KUKA KRL program: EPS_2_251825_SA31_A_20260116064112.src

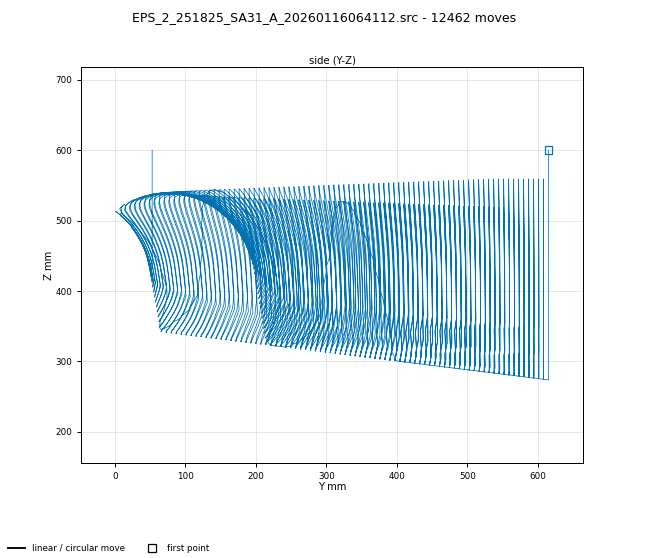
[picture p0: tool path of EPS_2_251825_SA31_A_20260116064112.src, 12462 of 12464 moves have a stored position in this frame; points joined in program order, loops and branches not executed]
&ACCESS RVP
&REL 4
&COMMENT QRS 19112012
&PARAM EDITMASK = *
DEF PART()
EXT BAS (BAS_COMMAND :IN,REAL :IN )
INT I
BAS (#INITMOV,0 )

;KUKA QRS Post kuka4.cps  Date:22-06-2017 !

File_ID=2978

QRS_PRE_INIT()

;Init var - Until changes are made in qrs_pre_init
Outlet_Square_prg=0
Inlet_1_Square_prg=0
Inlet_2_Square_prg=0
Inlet_3_Square_prg=0
Inlet_4_Square_prg=0
Inlet_5_Square_prg=0

Outlet_1={X 0.000, Y 535.490, Z 458.500, B 0.000, E1 0.000 }
Inlet_1={X 0.000, Y 538.340, Z 418.500, B 0.000, E1 227.000 }
Outlet_1_type=201
Inlet_1_type=201
;QRS#1=Sidecore dimensions
;QRS#2=200-8" PVC SDR 35
;QRS#3=200-8" PVC SDR 35
;QRS#4=
;QRS#5=
;QRS#6=
;QRS#7=
;QRS#8=
;QRS#9=12-08 PSX
;QRS#10=12-08 PSX
;QRS#11=
;QRS#12=
;QRS#13=
;QRS#14=
;QRS#15=
;QRS#16=1220x127x838 2,75'
;QRS#17=EPS Height
;QRS#18=559
;QRS#19=*
;QRS#20= UPDATED VERSION 22-06-2017
;QRS#21=*
Outlet_Square=0100
Inlet_1_Square=0100
Inlet_2_Square=0
Inlet_3_Square=0
Inlet_4_Square=0
Inlet_5_Square=0
Mill_Square=1
Outlet_Square_Prg=204
Inlet_1_Square_prg=204

QRS_INIT()

$ADVANCE=5

; T1
PTP {E1 173.626,E2 173.626}
PTP {X 0,Y 615.464,A -85,B 0,C 180,E1 173.626,E2 173.626,E3 0,E4 0,E5 0,E6 0}
QRS_SPEED_INIT()
LIN {X 0,Y 615.464,Z 600,A -85,B 0,C 180,E1 173.626,E2 173.626,E3 0,E4 0,E5 0,E6 0} C_VEL
LIN {X 0,Y 615.464,Z 283.872,A -85,B 0,C 180,E1 173.626,E2 173.626} C_VEL
LIN {X 0,Y 615.464,Z 275.69,A -85,B 0,C 180,E1 173.626,E2 173.626} C_VEL
LIN {X 0,Y 615.457,Z 273.69,A -85,B 0,C 180,E1 173.44,E2 173.44} C_VEL
LIN {X 0,Y 615.487,Z 273.682,A -85,B 0,C 180,E1 170.801,E2 170.801} C_VEL
LIN {X 0,Y 615.492,Z 273.695,A -85,B 0,C 180,E1 168.139,E2 168.139} C_VEL
LIN {X 0,Y 615.46,Z 273.694,A -85,B 0,C 180,E1 165.45,E2 165.45} C_VEL
LIN {X 0,Y 615.46,Z 273.695,A -85,B 0,C 180,E1 163.412,E2 163.412} C_VEL
LIN {X 0,Y 615.46,Z 273.694,A -85,B 0,C 180,E1 161.353,E2 161.353} C_VEL
LIN {X 0,Y 615.458,Z 273.694,A -85,B 0,C 180,E1 159.268,E2 159.268} C_VEL
LIN {X 0,Y 615.455,Z 273.694,A -85,B 0,C 180,E1 157.154,E2 157.154} C_VEL
LIN {X 0,Y 615.451,Z 273.693,A -85,B 0,C 180,E1 155.006,E2 155.006} C_VEL
LIN {X 0,Y 615.448,Z 273.691,A -85,B 0,C 180,E1 152.821,E2 152.821} C_VEL
LIN {X 0,Y 615.475,Z 273.685,A -85,B 0,C 180,E1 150.206,E2 150.206} C_VEL
LIN {X 0,Y 615.493,Z 273.696,A -85,B 0,C 180,E1 147.542,E2 147.542} C_VEL
LIN {X 0,Y 615.481,Z 273.698,A -85,B 0,C 180,E1 145.184,E2 145.184} C_VEL
LIN {X 0,Y 615.45,Z 273.695,A -85,B 0,C 180,E1 142.755,E2 142.755} C_VEL
LIN {X 0,Y 615.446,Z 273.69,A -85,B 0,C 180,E1 140.246,E2 140.246} C_VEL
LIN {X 0,Y 615.491,Z 273.685,A -85,B 0,C 180,E1 137.647,E2 137.647} C_VEL
LIN {X 0,Y 615.483,Z 273.699,A -85,B 0,C 180,E1 134.93,E2 134.93} C_VEL
LIN {X 0,Y 615.442,Z 273.694,A -85,B 0,C 180,E1 132.356,E2 132.356} C_VEL
LIN {X 0,Y 615.438,Z 273.692,A -85,B 0,C 180,E1 130.083,E2 130.083} C_VEL
LIN {X 0,Y 615.437,Z 273.692,A -85,B 0,C 180,E1 128.005,E2 128.005} C_VEL
LIN {X 0,Y 615.449,Z 273.69,A -85,B 0,C 180,E1 125.618,E2 125.618} C_VEL
LIN {X 0,Y 615.474,Z 273.689,A -85,B 0,C 180,E1 123.236,E2 123.236} C_VEL
LIN {X 0,Y 615.491,Z 273.693,A -85,B 0,C 180,E1 120.919,E2 120.919} C_VEL
LIN {X 0,Y 615.435,Z 273.695,A -85,B 0,C 180,E1 117.917,E2 117.917} C_VEL
LIN {X 0,Y 615.433,Z 273.693,A -85,B 0,C 180,E1 115.557,E2 115.557} C_VEL
LIN {X 0,Y 615.484,Z 273.69,A -85,B 0,C 180,E1 112.844,E2 112.844} C_VEL
LIN {X 0,Y 615.454,Z 273.698,A -85,B 0,C 180,E1 110.033,E2 110.033} C_VEL
LIN {X 0,Y 615.452,Z 273.698,A -85,B 0,C 180,E1 107.957,E2 107.957} C_VEL
LIN {X 0,Y 615.451,Z 273.698,A -85,B 0,C 180,E1 105.906,E2 105.906} C_VEL
LIN {X 0,Y 615.454,Z 273.698,A -85,B 0,C 180,E1 103.874,E2 103.874} C_VEL
LIN {X 0,Y 615.458,Z 273.699,A -85,B 0,C 180,E1 101.861,E2 101.861} C_VEL
LIN {X 0,Y 615.423,Z 273.696,A -85,B 0,C 180,E1 99.199,E2 99.199} C_VEL
LIN {X 0,Y 615.421,Z 273.697,A -85,B 0,C 180,E1 97.216,E2 97.216} C_VEL
LIN {X 0,Y 615.423,Z 273.697,A -85,B 0,C 180,E1 95.241,E2 95.241} C_VEL
LIN {X 0,Y 615.426,Z 273.697,A -85,B 0,C 180,E1 93.273,E2 93.273} C_VEL
LIN {X 0,Y 615.431,Z 273.698,A -85,B 0,C 180,E1 91.308,E2 91.308} C_VEL
LIN {X 0,Y 615.433,Z 273.699,A -85,B 0,C 180,E1 89.345,E2 89.345} C_VEL
LIN {X 0,Y 615.446,Z 273.699,A -85,B 0,C 180,E1 87.382,E2 87.382} C_VEL
LIN {X 0,Y 615.415,Z 273.697,A -85,B 0,C 180,E1 84.758,E2 84.758} C_VEL
LIN {X 0,Y 615.414,Z 273.698,A -85,B 0,C 180,E1 82.783,E2 82.783} C_VEL
LIN {X 0,Y 615.415,Z 273.698,A -85,B 0,C 180,E1 80.8,E2 80.8} C_VEL
LIN {X 0,Y 615.416,Z 273.699,A -85,B 0,C 180,E1 78.805,E2 78.805} C_VEL
LIN {X 0,Y 615.418,Z 273.699,A -85,B 0,C 180,E1 76.797,E2 76.797} C_VEL
LIN {X 0,Y 615.419,Z 273.699,A -85,B 0,C 180,E1 74.772,E2 74.772} C_VEL
LIN {X 0,Y 615.419,Z 273.699,A -85,B 0,C 180,E1 72.727,E2 72.727} C_VEL
LIN {X 0,Y 615.418,Z 273.699,A -85,B 0,C 180,E1 70.66,E2 70.66} C_VEL
LIN {X 0,Y 615.414,Z 273.699,A -85,B 0,C 180,E1 68.565,E2 68.565} C_VEL
LIN {X 0,Y 615.408,Z 273.7,A -85,B 0,C 180,E1 66.44,E2 66.44} C_VEL
LIN {X 0,Y 615.405,Z 273.7,A -85,B 0,C 180,E1 64.28,E2 64.28} C_VEL
LIN {X 0,Y 615.402,Z 273.7,A -85,B 0,C 180,E1 62.081,E2 62.081} C_VEL
LIN {X 0,Y 615.423,Z 273.873,A -85,B 0,C 180,E1 61.594,E2 61.594} C_VEL
LIN {X 0,Y 615.459,Z 291.447,A -85,B 0,C 180,E1 58.614,E2 58.614} C_VEL
LIN {X 0,Y 615.456,Z 305.727,A -85,B 0,C 180,E1 56.223,E2 56.223} C_VEL
LIN {X 0,Y 615.472,Z 308.215,A -85,B 0,C 180,E1 55.808,E2 55.808} C_VEL
LIN {X 0,Y 615.477,Z 415.41,A -85,B 0,C 180,E1 54.534,E2 54.534} C_VEL
LIN {X 0,Y 615.47,Z 427.253,A -85,B 0,C 180,E1 54.276,E2 54.276} C_VEL
LIN {X 0,Y 615.484,Z 439.785,A -85,B 0,C 180,E1 53.873,E2 53.873} C_VEL
LIN {X 0,Y 615.479,Z 451.084,A -85,B 0,C 180,E1 53.384,E2 53.384} C_VEL
LIN {X 0,Y 615.493,Z 462.353,A -85,B 0,C 180,E1 52.758,E2 52.758} C_VEL
LIN {X 0,Y 615.495,Z 473.289,A -85,B 0,C 180,E1 51.988,E2 51.988} C_VEL
LIN {X 0,Y 615.496,Z 481.209,A -85,B 0,C 180,E1 51.306,E2 51.306} C_VEL
LIN {X 0,Y 615.499,Z 489.826,A -85,B 0,C 180,E1 50.423,E2 50.423} C_VEL
LIN {X 0,Y 615.49,Z 496.02,A -85,B 0,C 180,E1 49.652,E2 49.652} C_VEL
LIN {X 0,Y 615.495,Z 503.395,A -85,B 0,C 180,E1 48.527,E2 48.527} C_VEL
LIN {X 0,Y 615.495,Z 507.948,A -85,B 0,C 180,E1 47.648,E2 47.648} C_VEL
LIN {X 0,Y 615.498,Z 511.617,A -85,B 0,C 180,E1 46.756,E2 46.756} C_VEL
LIN {X 0,Y 615.498,Z 514.488,A -85,B 0,C 180,E1 45.851,E2 45.851} C_VEL
LIN {X 0,Y 615.496,Z 516.585,A -85,B 0,C 180,E1 44.932,E2 44.932} C_VEL
LIN {X 0,Y 615.495,Z 517.891,A -85,B 0,C 180,E1 43.998,E2 43.998} C_VEL
LIN {X 0,Y 615.496,Z 518.372,A -85,B 0,C 180,E1 43.048,E2 43.048} C_VEL
LIN {X 0,Y 615.498,Z 518.018,A -85,B 0,C 180,E1 42.081,E2 42.081} C_VEL
LIN {X 0,Y 615.495,Z 516.78,A -85,B 0,C 180,E1 41.095,E2 41.095} C_VEL
LIN {X 0,Y 615.493,Z 513.618,A -85,B 0,C 180,E1 39.75,E2 39.75} C_VEL
LIN {X 0,Y 615.493,Z 508.935,A -85,B 0,C 180,E1 38.485,E2 38.485} C_VEL
LIN {X 0,Y 615.497,Z 503.671,A -85,B 0,C 180,E1 37.434,E2 37.434} C_VEL
LIN {X 0,Y 615.493,Z 497.261,A -85,B 0,C 180,E1 36.425,E2 36.425} C_VEL
LIN {X 0,Y 615.493,Z 489.182,A -85,B 0,C 180,E1 35.415,E2 35.415} C_VEL
LIN {X 0,Y 615.494,Z 478.595,A -85,B 0,C 180,E1 34.362,E2 34.362} C_VEL
LIN {X 0,Y 615.497,Z 468.094,A -85,B 0,C 180,E1 33.535,E2 33.535} C_VEL
LIN {X 0,Y 615.46,Z 457.245,A -85,B 0,C 180,E1 32.848,E2 32.848} C_VEL
LIN {X 0,Y 615.493,Z 445.048,A -85,B 0,C 180,E1 32.25,E2 32.25} C_VEL
LIN {X 0,Y 615.466,Z 433.199,A -85,B 0,C 180,E1 31.808,E2 31.808} C_VEL
LIN {X 0,Y 615.439,Z 419.96,A -85,B 0,C 180,E1 31.459,E2 31.459} C_VEL
LIN {X 0,Y 615.434,Z 406.25,A -85,B 0,C 180,E1 31.249,E2 31.249} C_VEL
LIN {X 0,Y 615.497,Z 308.14,A -85,B 0,C 180,E1 30.091,E2 30.091} C_VEL
LIN {X 0,Y 615.466,Z 291.844,A -85,B 0,C 180,E1 27.363,E2 27.363} C_VEL
LIN {X 0,Y 615.481,Z 275.707,A -85,B 0,C 180,E1 24.632,E2 24.632} C_VEL
LIN {X 0,Y 615.473,Z 273.688,A -85,B 0,C 180,E1 24.273,E2 24.273} C_VEL
LIN {X 0,Y 615.474,Z 273.686,A -85,B 0,C 180,E1 22.137,E2 22.137} C_VEL
LIN {X 0,Y 615.48,Z 273.685,A -85,B 0,C 180,E1 19.338,E2 19.338} C_VEL
LIN {X 0,Y 615.482,Z 273.697,A -85,B 0,C 180,E1 16.429,E2 16.429} C_VEL
LIN {X 0,Y 615.474,Z 273.686,A -85,B 0,C 180,E1 13.875,E2 13.875} C_VEL
LIN {X 0,Y 615.486,Z 273.682,A -85,B 0,C 180,E1 11.193,E2 11.193} C_VEL
LIN {X 0,Y 615.483,Z 273.696,A -85,B 0,C 180,E1 8.537,E2 8.537} C_VEL
LIN {X 0,Y 615.475,Z 273.693,A -85,B 0,C 180,E1 5.899,E2 5.899} C_VEL
LIN {X 0,Y 615.485,Z 273.681,A -85,B 0,C 180,E1 3.273,E2 3.273} C_VEL
LIN {X 0,Y 615.477,Z 273.687,A -85,B 0,C 180,E1 0.654,E2 0.654} C_VEL
LIN {X 0,Y 615.497,Z 273.7,A -85,B 0,C 180,E1 -1.963,E2 -1.963} C_VEL
LIN {X 0,Y 615.472,Z 273.69,A -85,B 0,C 180,E1 -4.585,E2 -4.585} C_VEL
LIN {X 0,Y 615.486,Z 273.681,A -85,B 0,C 180,E1 -7.216,E2 -7.216} C_VEL
LIN {X 0,Y 615.479,Z 273.691,A -85,B 0,C 180,E1 -9.862,E2 -9.862} C_VEL
LIN {X 0,Y 615.479,Z 273.697,A -85,B 0,C 180,E1 -12.53,E2 -12.53} C_VEL
LIN {X 0,Y 615.478,Z 273.683,A -85,B 0,C 180,E1 -15.226,E2 -15.226} C_VEL
LIN {X 0,Y 615.478,Z 273.687,A -85,B 0,C 180,E1 -17.957,E2 -17.957} C_VEL
LIN {X 0,Y 615.483,Z 273.699,A -85,B 0,C 180,E1 -20.731,E2 -20.731} C_VEL
LIN {X 0,Y 615.48,Z 273.682,A -85,B 0,C 180,E1 -23.557,E2 -23.557} C_VEL
LIN {X 0,Y 615.481,Z 273.692,A -85,B 0,C 180,E1 -26.444,E2 -26.444} C_VEL
LIN {X 0,Y 615.486,Z 273.695,A -85,B 0,C 180,E1 -28.658,E2 -28.658} C_VEL
LIN {X 0,Y 615.481,Z 273.698,A -85,B 0,C 180,E1 -31.085,E2 -31.085} C_VEL
LIN {X 0,Y 615.489,Z 273.68,A -85,B 0,C 180,E1 -34.022,E2 -34.022} C_VEL
LIN {X 0,Y 615.483,Z 273.696,A -85,B 0,C 180,E1 -36.936,E2 -36.936} C_VEL
LIN {X 0,Y 615.47,Z 273.689,A -85,B 0,C 180,E1 -39.752,E2 -39.752} C_VEL
LIN {X 0,Y 615.493,Z 273.679,A -85,B 0,C 180,E1 -42.353,E2 -42.353} C_VEL
LIN {X 0,Y 615.482,Z 273.692,A -85,B 0,C 180,E1 -45.069,E2 -45.069} C_VEL
LIN {X 0,Y 615.47,Z 273.691,A -85,B 0,C 180,E1 -47.922,E2 -47.922} C_VEL
LIN {X 0,Y 615.471,Z 273.686,A -85,B 0,C 180,E1 -50.248,E2 -50.248} C_VEL
LIN {X 0,Y 615.482,Z 273.686,A -85,B 0,C 180,E1 -53.064,E2 -53.064} C_VEL
LIN {X 0,Y 615.479,Z 273.695,A -85,B 0,C 180,E1 -55.977,E2 -55.977} C_VEL
LIN {X 0,Y 615.469,Z 273.69,A -85,B 0,C 180,E1 -58.313,E2 -58.313} C_VEL
LIN {X 0,Y 615.469,Z 273.687,A -85,B 0,C 180,E1 -60.593,E2 -60.593} C_VEL
LIN {X 0,Y 615.486,Z 273.681,A -85,B 0,C 180,E1 -62.956,E2 -62.956} C_VEL
LIN {X 0,Y 615.481,Z 273.692,A -85,B 0,C 180,E1 -65.727,E2 -65.727} C_VEL
LIN {X 0,Y 615.487,Z 273.753,A -85,B 0,C 180,E1 -67.437,E2 -67.437} C_VEL
LIN {X 0,Y 615.455,Z 293.69,A -85,B 0,C 180,E1 -70.14,E2 -70.14} C_VEL
LIN {X 0,Y 615.472,Z 313.075,A -85,B 0,C 180,E1 -72.729,E2 -72.729} C_VEL
LIN {X 0,Y 615.493,Z 334.915,A -85,B 0,C 180,E1 -75.606,E2 -75.606} C_VEL
LIN {X 0,Y 615.471,Z 346.466,A -85,B 0,C 180,E1 -77.113,E2 -77.113} C_VEL
LIN {X 0,Y 615.457,Z 454.82,A -85,B 0,C 180,E1 -78.41,E2 -78.41} C_VEL
LIN {X 0,Y 615.456,Z 467.338,A -85,B 0,C 180,E1 -78.681,E2 -78.681} C_VEL
LIN {X 0,Y 615.483,Z 480.687,A -85,B 0,C 180,E1 -79.115,E2 -79.115} C_VEL
LIN {X 0,Y 615.492,Z 492.47,A -85,B 0,C 180,E1 -79.639,E2 -79.639} C_VEL
LIN {X 0,Y 615.483,Z 503.991,A -85,B 0,C 180,E1 -80.303,E2 -80.303} C_VEL
LIN {X 0,Y 615.499,Z 514.337,A -85,B 0,C 180,E1 -81.05,E2 -81.05} C_VEL
LIN {X 0,Y 615.497,Z 522.688,A -85,B 0,C 180,E1 -81.794,E2 -81.794} C_VEL
LIN {X 0,Y 615.498,Z 530.603,A -85,B 0,C 180,E1 -82.619,E2 -82.619} C_VEL
LIN {X 0,Y 615.491,Z 538.202,A -85,B 0,C 180,E1 -83.608,E2 -83.608} C_VEL
LIN {X 0,Y 615.498,Z 545.203,A -85,B 0,C 180,E1 -84.759,E2 -84.759} C_VEL
LIN {X 0,Y 615.493,Z 549.85,A -85,B 0,C 180,E1 -85.743,E2 -85.743} C_VEL
LIN {X 0,Y 615.494,Z 553.398,A -85,B 0,C 180,E1 -86.727,E2 -86.727} C_VEL
LIN {X 0,Y 615.497,Z 555.232,A -85,B 0,C 180,E1 -87.382,E2 -87.382} C_VEL
LIN {X 0,Y 615.497,Z 556.607,A -85,B 0,C 180,E1 -88.037,E2 -88.037} C_VEL
LIN {X 0,Y 615.496,Z 558.173,A -85,B 0,C 180,E1 -89.345,E2 -89.345} C_VEL
LIN {X 0,Y 615.494,Z 558.389,A -85,B 0,C 180,E1 -90,E2 -90} C_VEL
LIN {X 0,Y 615.495,Z 557.58,A -85,B 0,C 180,E1 -91.308,E2 -91.308} C_VEL
LIN {X 0,Y 615.497,Z 556.609,A -85,B 0,C 180,E1 -91.963,E2 -91.963} C_VEL
LIN {X 0,Y 615.497,Z 555.234,A -85,B 0,C 180,E1 -92.617,E2 -92.617} C_VEL
LIN {X 0,Y 615.496,Z 552.351,A -85,B 0,C 180,E1 -93.6,E2 -93.6} C_VEL
LIN {X 0,Y 615.498,Z 548.443,A -85,B 0,C 180,E1 -94.584,E2 -94.584} C_VEL
LIN {X 0,Y 615.499,Z 543.407,A -85,B 0,C 180,E1 -95.569,E2 -95.569} C_VEL
LIN {X 0,Y 615.49,Z 536.913,A -85,B 0,C 180,E1 -96.578,E2 -96.578} C_VEL
LIN {X 0,Y 615.497,Z 529.137,A -85,B 0,C 180,E1 -97.545,E2 -97.545} C_VEL
LIN {X 0,Y 615.498,Z 519.262,A -85,B 0,C 180,E1 -98.536,E2 -98.536} C_VEL
LIN {X 0,Y 615.495,Z 508.872,A -85,B 0,C 180,E1 -99.364,E2 -99.364} C_VEL
LIN {X 0,Y 615.482,Z 498.584,A -85,B 0,C 180,E1 -100.028,E2 -100.028} C_VEL
LIN {X 0,Y 615.495,Z 487.144,A -85,B 0,C 180,E1 -100.616,E2 -100.616} C_VEL
LIN {X 0,Y 615.467,Z 475.366,A -85,B 0,C 180,E1 -101.077,E2 -101.077} C_VEL
LIN {X 0,Y 615.455,Z 462.267,A -85,B 0,C 180,E1 -101.443,E2 -101.443} C_VEL
LIN {X 0,Y 615.461,Z 448.986,A -85,B 0,C 180,E1 -101.673,E2 -101.673} C_VEL
LIN {X 0,Y 615.471,Z 346.472,A -85,B 0,C 180,E1 -102.886,E2 -102.886} C_VEL
LIN {X 0,Y 615.455,Z 325.994,A -85,B 0,C 180,E1 -105.566,E2 -105.566} C_VEL
LIN {X 0,Y 615.481,Z 305.476,A -85,B 0,C 180,E1 -108.281,E2 -108.281} C_VEL
LIN {X 0,Y 615.468,Z 283.348,A -85,B 0,C 180,E1 -111.256,E2 -111.256} C_VEL
LIN {X 0,Y 615.489,Z 273.682,A -85,B 0,C 180,E1 -112.594,E2 -112.594} C_VEL
LIN {X 0,Y 615.485,Z 273.681,A -85,B 0,C 180,E1 -114.991,E2 -114.991} C_VEL
LIN {X 0,Y 615.482,Z 273.699,A -85,B 0,C 180,E1 -117.915,E2 -117.915} C_VEL
LIN {X 0,Y 615.485,Z 273.682,A -85,B 0,C 180,E1 -120.919,E2 -120.919} C_VEL
LIN {X 0,Y 615.473,Z 273.686,A -85,B 0,C 180,E1 -123.532,E2 -123.532} C_VEL
LIN {X 0,Y 615.487,Z 273.696,A -85,B 0,C 180,E1 -126.424,E2 -126.424} C_VEL
LIN {X 0,Y 615.48,Z 273.684,A -85,B 0,C 180,E1 -129.061,E2 -129.061} C_VEL
LIN {X 0,Y 615.492,Z 273.68,A -85,B 0,C 180,E1 -131.473,E2 -131.473} C_VEL
LIN {X 0,Y 615.477,Z 273.693,A -85,B 0,C 180,E1 -134.15,E2 -134.15} C_VEL
LIN {X 0,Y 615.476,Z 273.691,A -85,B 0,C 180,E1 -136.953,E2 -136.953} C_VEL
LIN {X 0,Y 615.481,Z 273.683,A -85,B 0,C 180,E1 -139.393,E2 -139.393} C_VEL
LIN {X 0,Y 615.482,Z 273.684,A -85,B 0,C 180,E1 -141.988,E2 -141.988} C_VEL
LIN {X 0,Y 615.479,Z 273.692,A -85,B 0,C 180,E1 -144.383,E2 -144.383} C_VEL
LIN {X 0,Y 615.484,Z 273.702,A -85,B 0,C 180,E1 -146.764,E2 -146.764} C_VEL
LIN {X 0,Y 615.48,Z 273.697,A -85,B 0,C 180,E1 -149.08,E2 -149.08} C_VEL
LIN {X 0,Y 615.47,Z 273.688,A -85,B 0,C 180,E1 -151.551,E2 -151.551} C_VEL
LIN {X 0,Y 615.49,Z 273.682,A -85,B 0,C 180,E1 -154.284,E2 -154.284} C_VEL
LIN {X 0,Y 615.484,Z 273.701,A -85,B 0,C 180,E1 -157.155,E2 -157.155} C_VEL
LIN {X 0,Y 615.471,Z 273.685,A -85,B 0,C 180,E1 -159.967,E2 -159.967} C_VEL
LIN {X 0,Y 615.483,Z 273.687,A -85,B 0,C 180,E1 -162.729,E2 -162.729} C_VEL
LIN {X 0,Y 615.482,Z 273.699,A -85,B 0,C 180,E1 -165.451,E2 -165.451} C_VEL
LIN {X 0,Y 615.464,Z 273.687,A -85,B 0,C 180,E1 -168.139,E2 -168.139} C_VEL
LIN {X 0,Y 615.493,Z 273.682,A -85,B 0,C 180,E1 -170.801,E2 -170.801} C_VEL
LIN {X 0,Y 615.494,Z 273.697,A -85,B 0,C 180,E1 -173.444,E2 -173.444} C_VEL
LIN {X 0,Y 615.464,Z 273.693,A -85,B 0,C 180,E1 -176.071,E2 -176.071} C_VEL
LIN {X 0,Y 615.474,Z 273.684,A -85,B 0,C 180,E1 -178.692,E2 -178.692} C_VEL
LIN {X 0,Y 615.488,Z 273.687,A -85,B 0,C 180,E1 -181.309,E2 -181.309} C_VEL
LIN {X 0,Y 615.483,Z 273.7,A -85,B 0,C 180,E1 -183.929,E2 -183.929} C_VEL
LIN {X 0,Y 615.457,Z 273.69,A -85,B 0,C 180,E1 -186.56,E2 -186.56} C_VEL
LIN {X 0,Y 614.8,Z 273.833,A -85,B 0,C 180,E1 -187.106,E2 -187.106} C_VEL
LIN {X 0,Y 611.98,Z 274.258,A -85,B 0,C 180,E1 -187.992,E2 -187.992} C_VEL
LIN {X 0,Y 609.59,Z 274.561,A -85,B 0,C 180,E1 -188.705,E2 -188.705} C_VEL
LIN {X 0,Y 608.552,Z 274.677,A -85,B 0,C 180,E1 -189.255,E2 -189.255} C_VEL
LIN {X 0,Y 608.461,Z 274.688,A -85,B 0,C 180,E1 -189.441,E2 -189.441} C_VEL
LIN {X 0,Y 608.46,Z 274.696,A -85,B 0,C 180,E1 -192,E2 -192} C_VEL
LIN {X 0,Y 608.426,Z 274.692,A -85,B 0,C 180,E1 -194.722,E2 -194.722} C_VEL
LIN {X 0,Y 608.426,Z 274.691,A -85,B 0,C 180,E1 -196.785,E2 -196.785} C_VEL
LIN {X 0,Y 608.442,Z 274.689,A -85,B 0,C 180,E1 -199.571,E2 -199.571} C_VEL
LIN {X 0,Y 608.454,Z 274.695,A -85,B 0,C 180,E1 -202.477,E2 -202.477} C_VEL
LIN {X 0,Y 608.444,Z 274.696,A -85,B 0,C 180,E1 -204.572,E2 -204.572} C_VEL
LIN {X 0,Y 608.427,Z 274.69,A -85,B 0,C 180,E1 -207.199,E2 -207.199} C_VEL
LIN {X 0,Y 608.46,Z 274.686,A -85,B 0,C 180,E1 -209.78,E2 -209.78} C_VEL
LIN {X 0,Y 608.465,Z 274.695,A -85,B 0,C 180,E1 -212.524,E2 -212.524} C_VEL
LIN {X 0,Y 608.421,Z 274.692,A -85,B 0,C 180,E1 -215.28,E2 -215.28} C_VEL
LIN {X 0,Y 608.448,Z 274.687,A -85,B 0,C 180,E1 -217.748,E2 -217.748} C_VEL
LIN {X 0,Y 608.443,Z 274.691,A -85,B 0,C 180,E1 -220.329,E2 -220.329} C_VEL
LIN {X 0,Y 608.45,Z 274.691,A -85,B 0,C 180,E1 -223.308,E2 -223.308} C_VEL
LIN {X 0,Y 608.44,Z 274.688,A -85,B 0,C 180,E1 -226.129,E2 -226.129} C_VEL
LIN {X 0,Y 608.461,Z 274.693,A -85,B 0,C 180,E1 -228.825,E2 -228.825} C_VEL
LIN {X 0,Y 608.434,Z 274.69,A -85,B 0,C 180,E1 -231.765,E2 -231.765} C_VEL
LIN {X 0,Y 608.429,Z 274.69,A -85,B 0,C 180,E1 -233.958,E2 -233.958} C_VEL
LIN {X 0,Y 608.427,Z 274.69,A -85,B 0,C 180,E1 -236.328,E2 -236.328} C_VEL
LIN {X 0,Y 608.442,Z 274.69,A -85,B 0,C 180,E1 -238.734,E2 -238.734} C_VEL
LIN {X 0,Y 608.427,Z 274.695,A -85,B 0,C 180,E1 -241.733,E2 -241.733} C_VEL
LIN {X 0,Y 608.428,Z 274.69,A -85,B 0,C 180,E1 -244.289,E2 -244.289} C_VEL
LIN {X 0,Y 608.429,Z 274.691,A -85,B 0,C 180,E1 -246.876,E2 -246.876} C_VEL
LIN {X 0,Y 608.45,Z 274.696,A -85,B 0,C 180,E1 -249.726,E2 -249.726} C_VEL
LIN {X 0,Y 608.429,Z 274.698,A -85,B 0,C 180,E1 -251.828,E2 -251.828} C_VEL
LIN {X 0,Y 608.443,Z 274.696,A -85,B 0,C 180,E1 -253.906,E2 -253.906} C_VEL
LIN {X 0,Y 608.436,Z 274.696,A -85,B 0,C 180,E1 -255.998,E2 -255.998} C_VEL
LIN {X 0,Y 608.409,Z 274.692,A -85,B 0,C 180,E1 -258.675,E2 -258.675} C_VEL
LIN {X 0,Y 608.43,Z 274.691,A -85,B 0,C 180,E1 -261.364,E2 -261.364} C_VEL
LIN {X 0,Y 608.455,Z 274.698,A -85,B 0,C 180,E1 -264.033,E2 -264.033} C_VEL
LIN {X 0,Y 608.399,Z 274.695,A -85,B 0,C 180,E1 -266.689,E2 -266.689} C_VEL
LIN {X 0,Y 608.422,Z 274.693,A -85,B 0,C 180,E1 -268.677,E2 -268.677} C_VEL
LIN {X 0,Y 608.412,Z 274.695,A -85,B 0,C 180,E1 -270.662,E2 -270.662} C_VEL
LIN {X 0,Y 608.439,Z 274.692,A -85,B 0,C 180,E1 -272.649,E2 -272.649} C_VEL
LIN {X 0,Y 608.402,Z 274.693,A -85,B 0,C 180,E1 -275.303,E2 -275.303} C_VEL
LIN {X 0,Y 608.4,Z 274.693,A -85,B 0,C 180,E1 -277.301,E2 -277.301} C_VEL
LIN {X 0,Y 608.417,Z 274.694,A -85,B 0,C 180,E1 -279.978,E2 -279.978} C_VEL
LIN {X 0,Y 608.458,Z 274.694,A -85,B 0,C 180,E1 -282.678,E2 -282.678} C_VEL
LIN {X 0,Y 608.385,Z 274.695,A -85,B 0,C 180,E1 -285.408,E2 -285.408} C_VEL
LIN {X 0,Y 608.393,Z 274.694,A -85,B 0,C 180,E1 -287.479,E2 -287.479} C_VEL
LIN {X 0,Y 608.391,Z 274.694,A -85,B 0,C 180,E1 -289.573,E2 -289.573} C_VEL
LIN {X 0,Y 608.38,Z 274.695,A -85,B 0,C 180,E1 -291.695,E2 -291.695} C_VEL
LIN {X 0,Y 608.389,Z 274.695,A -85,B 0,C 180,E1 -294.133,E2 -294.133} C_VEL
LIN {X 0,Y 608.42,Z 274.7,A -85,B 0,C 180,E1 -296.776,E2 -296.776} C_VEL
LIN {X 0,Y 608.386,Z 274.697,A -85,B 0,C 180,E1 -298.314,E2 -298.314} C_VEL
LIN {X 0,Y 608.485,Z 289.811,A -85,B 0,C 180,E1 -300.904,E2 -300.904} C_VEL
LIN {X 0,Y 608.448,Z 306.21,A -85,B 0,C 180,E1 -303.672,E2 -303.672} C_VEL
LIN {X 0,Y 608.46,Z 308.488,A -85,B 0,C 180,E1 -304.044,E2 -304.044} C_VEL
LIN {X 0,Y 608.545,Z 415.653,A -85,B 0,C 180,E1 -305.334,E2 -305.334} C_VEL
LIN {X 0,Y 608.522,Z 429.543,A -85,B 0,C 180,E1 -305.653,E2 -305.653} C_VEL
LIN {X 0,Y 608.507,Z 442.198,A -85,B 0,C 180,E1 -306.088,E2 -306.088} C_VEL
LIN {X 0,Y 608.5,Z 453.351,A -85,B 0,C 180,E1 -306.602,E2 -306.602} C_VEL
LIN {X 0,Y 608.499,Z 464.515,A -85,B 0,C 180,E1 -307.257,E2 -307.257} C_VEL
LIN {X 0,Y 608.484,Z 474.623,A -85,B 0,C 180,E1 -307.993,E2 -307.993} C_VEL
LIN {X 0,Y 608.459,Z 483.584,A -85,B 0,C 180,E1 -308.801,E2 -308.801} C_VEL
LIN {X 0,Y 608.47,Z 491.584,A -85,B 0,C 180,E1 -309.654,E2 -309.654} C_VEL
LIN {X 0,Y 608.435,Z 499.7,A -85,B 0,C 180,E1 -310.74,E2 -310.74} C_VEL
LIN {X 0,Y 608.445,Z 506.352,A -85,B 0,C 180,E1 -311.868,E2 -311.868} C_VEL
LIN {X 0,Y 608.438,Z 511.268,A -85,B 0,C 180,E1 -312.961,E2 -312.961} C_VEL
LIN {X 0,Y 608.423,Z 515.446,A -85,B 0,C 180,E1 -314.26,E2 -314.26} C_VEL
LIN {X 0,Y 608.419,Z 517.436,A -85,B 0,C 180,E1 -315.2,E2 -315.2} C_VEL
LIN {X 0,Y 608.429,Z 518.603,A -85,B 0,C 180,E1 -316.126,E2 -316.126} C_VEL
LIN {X 0,Y 608.436,Z 519,A -85,B 0,C 180,E1 -317.038,E2 -317.038} C_VEL
LIN {X 0,Y 608.425,Z 518.623,A -85,B 0,C 180,E1 -317.935,E2 -317.935} C_VEL
LIN {X 0,Y 608.432,Z 517.55,A -85,B 0,C 180,E1 -318.821,E2 -318.821} C_VEL
LIN {X 0,Y 608.438,Z 514.651,A -85,B 0,C 180,E1 -320.127,E2 -320.127} C_VEL
LIN {X 0,Y 608.435,Z 511.527,A -85,B 0,C 180,E1 -321.059,E2 -321.059} C_VEL
LIN {X 0,Y 608.438,Z 506.2,A -85,B 0,C 180,E1 -322.251,E2 -322.251} C_VEL
LIN {X 0,Y 608.449,Z 500.099,A -85,B 0,C 180,E1 -323.291,E2 -323.291} C_VEL
LIN {X 0,Y 608.449,Z 492.379,A -85,B 0,C 180,E1 -324.338,E2 -324.338} C_VEL
LIN {X 0,Y 608.469,Z 484.982,A -85,B 0,C 180,E1 -325.151,E2 -325.151} C_VEL
LIN {X 0,Y 608.471,Z 476.652,A -85,B 0,C 180,E1 -325.93,E2 -325.93} C_VEL
LIN {X 0,Y 608.476,Z 466.142,A -85,B 0,C 180,E1 -326.726,E2 -326.726} C_VEL
LIN {X 0,Y 608.481,Z 454.916,A -85,B 0,C 180,E1 -327.404,E2 -327.404} C_VEL
LIN {X 0,Y 608.516,Z 443.264,A -85,B 0,C 180,E1 -327.957,E2 -327.957} C_VEL
LIN {X 0,Y 608.513,Z 431.009,A -85,B 0,C 180,E1 -328.395,E2 -328.395} C_VEL
LIN {X 0,Y 608.5,Z 418.028,A -85,B 0,C 180,E1 -328.713,E2 -328.713} C_VEL
LIN {X 0,Y 608.496,Z 398.865,A -85,B 0,C 180,E1 -328.975,E2 -328.975} C_VEL
LIN {X 0,Y 608.468,Z 308.395,A -85,B 0,C 180,E1 -330.051,E2 -330.051} C_VEL
LIN {X 0,Y 608.466,Z 292.117,A -85,B 0,C 180,E1 -332.795,E2 -332.795} C_VEL
LIN {X 0,Y 608.48,Z 276.69,A -85,B 0,C 180,E1 -335.43,E2 -335.43} C_VEL
LIN {X 0,Y 608.459,Z 274.688,A -85,B 0,C 180,E1 -335.805,E2 -335.805} C_VEL
LIN {X 0,Y 608.462,Z 274.685,A -85,B 0,C 180,E1 -338.308,E2 -338.308} C_VEL
LIN {X 0,Y 608.473,Z 274.695,A -85,B 0,C 180,E1 -341.284,E2 -341.284} C_VEL
LIN {X 0,Y 608.453,Z 274.689,A -85,B 0,C 180,E1 -343.906,E2 -343.906} C_VEL
LIN {X 0,Y 608.459,Z 274.686,A -85,B 0,C 180,E1 -346.643,E2 -346.643} C_VEL
LIN {X 0,Y 608.465,Z 274.692,A -85,B 0,C 180,E1 -349.35,E2 -349.35} C_VEL
LIN {X 0,Y 608.468,Z 274.689,A -85,B 0,C 180,E1 -352.033,E2 -352.033} C_VEL
LIN {X 0,Y 608.467,Z 274.685,A -85,B 0,C 180,E1 -354.698,E2 -354.698} C_VEL
LIN {X 0,Y 608.471,Z 274.687,A -85,B 0,C 180,E1 -357.352,E2 -357.352} C_VEL
LIN {X 0,Y 608.477,Z 274.694,A -85,B 0,C 180,E1 -360,E2 -360} C_VEL
LIN {X 0,Y 608.463,Z 274.687,A -85,B 0,C 180,E1 -362.648,E2 -362.648} C_VEL
LIN {X 0,Y 608.468,Z 274.685,A -85,B 0,C 180,E1 -365.302,E2 -365.302} C_VEL
LIN {X 0,Y 608.473,Z 274.691,A -85,B 0,C 180,E1 -367.967,E2 -367.967} C_VEL
LIN {X 0,Y 608.456,Z 274.691,A -85,B 0,C 180,E1 -370.65,E2 -370.65} C_VEL
LIN {X 0,Y 608.458,Z 274.685,A -85,B 0,C 180,E1 -373.356,E2 -373.356} C_VEL
LIN {X 0,Y 608.458,Z 274.691,A -85,B 0,C 180,E1 -376.094,E2 -376.094} C_VEL
LIN {X 0,Y 608.456,Z 274.691,A -85,B 0,C 180,E1 -378.87,E2 -378.87} C_VEL
LIN {X 0,Y 608.459,Z 274.685,A -85,B 0,C 180,E1 -381.692,E2 -381.692} C_VEL
LIN {X 0,Y 608.447,Z 274.696,A -85,B 0,C 180,E1 -384.571,E2 -384.571} C_VEL
LIN {X 0,Y 608.471,Z 274.688,A -85,B 0,C 180,E1 -387.206,E2 -387.206} C_VEL
LIN {X 0,Y 608.466,Z 274.685,A -85,B 0,C 180,E1 -389.971,E2 -389.971} C_VEL
LIN {X 0,Y 608.451,Z 274.696,A -85,B 0,C 180,E1 -392.88,E2 -392.88} C_VEL
LIN {X 0,Y 608.432,Z 274.696,A -85,B 0,C 180,E1 -395.278,E2 -395.278} C_VEL
LIN {X 0,Y 608.466,Z 274.686,A -85,B 0,C 180,E1 -397.747,E2 -397.747} C_VEL
LIN {X 0,Y 608.446,Z 274.687,A -85,B 0,C 180,E1 -400.328,E2 -400.328} C_VEL
LIN {X 0,Y 608.477,Z 274.695,A -85,B 0,C 180,E1 -403.309,E2 -403.309} C_VEL
LIN {X 0,Y 608.458,Z 274.687,A -85,B 0,C 180,E1 -406.129,E2 -406.129} C_VEL
LIN {X 0,Y 608.455,Z 274.687,A -85,B 0,C 180,E1 -408.823,E2 -408.823} C_VEL
LIN {X 0,Y 608.459,Z 274.694,A -85,B 0,C 180,E1 -411.761,E2 -411.761} C_VEL
LIN {X 0,Y 608.444,Z 274.694,A -85,B 0,C 180,E1 -413.955,E2 -413.955} C_VEL
LIN {X 0,Y 608.445,Z 274.69,A -85,B 0,C 180,E1 -416.328,E2 -416.328} C_VEL
LIN {X 0,Y 608.446,Z 274.687,A -85,B 0,C 180,E1 -418.733,E2 -418.733} C_VEL
LIN {X 0,Y 608.471,Z 274.687,A -85,B 0,C 180,E1 -421.381,E2 -421.381} C_VEL
LIN {X 0,Y 608.438,Z 274.7,A -85,B 0,C 180,E1 -423.964,E2 -423.964} C_VEL
LIN {X 0,Y 608.464,Z 274.696,A -85,B 0,C 180,E1 -426.155,E2 -426.155} C_VEL
LIN {X 0,Y 608.507,Z 274.819,A -85,B 0,C 180,E1 -427.312,E2 -427.312} C_VEL
LIN {X 0,Y 608.524,Z 292.405,A -85,B 0,C 180,E1 -429.728,E2 -429.728} C_VEL
LIN {X 0,Y 608.51,Z 311.822,A -85,B 0,C 180,E1 -432.351,E2 -432.351} C_VEL
LIN {X 0,Y 608.496,Z 332.533,A -85,B 0,C 180,E1 -435.109,E2 -435.109} C_VEL
LIN {X 0,Y 608.454,Z 346.611,A -85,B 0,C 180,E1 -436.962,E2 -436.962} C_VEL
LIN {X 0,Y 608.566,Z 386.467,A -85,B 0,C 180,E1 -437.452,E2 -437.452} C_VEL
LIN {X 0,Y 608.522,Z 454.93,A -85,B 0,C 180,E1 -438.276,E2 -438.276} C_VEL
LIN {X 0,Y 608.491,Z 468.205,A -85,B 0,C 180,E1 -438.571,E2 -438.571} C_VEL
LIN {X 0,Y 608.511,Z 480.649,A -85,B 0,C 180,E1 -438.983,E2 -438.983} C_VEL
LIN {X 0,Y 608.514,Z 492.629,A -85,B 0,C 180,E1 -439.519,E2 -439.519} C_VEL
LIN {X 0,Y 608.471,Z 504.192,A -85,B 0,C 180,E1 -440.191,E2 -440.191} C_VEL
LIN {X 0,Y 608.485,Z 514.589,A -85,B 0,C 180,E1 -440.945,E2 -440.945} C_VEL
LIN {X 0,Y 608.459,Z 522.999,A -85,B 0,C 180,E1 -441.698,E2 -441.698} C_VEL
LIN {X 0,Y 608.471,Z 530.957,A -85,B 0,C 180,E1 -442.534,E2 -442.534} C_VEL
LIN {X 0,Y 608.437,Z 538.297,A -85,B 0,C 180,E1 -443.486,E2 -443.486} C_VEL
LIN {X 0,Y 608.45,Z 543.864,A -85,B 0,C 180,E1 -444.365,E2 -444.365} C_VEL
LIN {X 0,Y 608.432,Z 548.948,A -85,B 0,C 180,E1 -445.362,E2 -445.362} C_VEL
LIN {X 0,Y 608.449,Z 552.895,A -85,B 0,C 180,E1 -446.357,E2 -446.357} C_VEL
LIN {X 0,Y 608.425,Z 555.808,A -85,B 0,C 180,E1 -447.351,E2 -447.351} C_VEL
LIN {X 0,Y 608.442,Z 557.201,A -85,B 0,C 180,E1 -448.014,E2 -448.014} C_VEL
LIN {X 0,Y 608.438,Z 558.783,A -85,B 0,C 180,E1 -449.338,E2 -449.338} C_VEL
LIN {X 0,Y 608.434,Z 559,A -85,B 0,C 180,E1 -450,E2 -450} C_VEL
LIN {X 0,Y 608.448,Z 558.184,A -85,B 0,C 180,E1 -451.323,E2 -451.323} C_VEL
LIN {X 0,Y 608.442,Z 557.202,A -85,B 0,C 180,E1 -451.985,E2 -451.985} C_VEL
LIN {X 0,Y 608.425,Z 555.81,A -85,B 0,C 180,E1 -452.648,E2 -452.648} C_VEL
LIN {X 0,Y 608.449,Z 552.898,A -85,B 0,C 180,E1 -453.642,E2 -453.642} C_VEL
LIN {X 0,Y 608.432,Z 548.952,A -85,B 0,C 180,E1 -454.637,E2 -454.637} C_VEL
LIN {X 0,Y 608.437,Z 542.879,A -85,B 0,C 180,E1 -455.8,E2 -455.8} C_VEL
LIN {X 0,Y 608.461,Z 536.238,A -85,B 0,C 180,E1 -456.799,E2 -456.799} C_VEL
LIN {X 0,Y 608.455,Z 527.993,A -85,B 0,C 180,E1 -457.8,E2 -457.8} C_VEL
LIN {X 0,Y 608.477,Z 517.604,A -85,B 0,C 180,E1 -458.803,E2 -458.803} C_VEL
LIN {X 0,Y 608.488,Z 506.754,A -85,B 0,C 180,E1 -459.641,E2 -459.641} C_VEL
LIN {X 0,Y 608.491,Z 495.782,A -85,B 0,C 180,E1 -460.312,E2 -460.312} C_VEL
LIN {X 0,Y 608.534,Z 483.807,A -85,B 0,C 180,E1 -460.888,E2 -460.888} C_VEL
LIN {X 0,Y 608.505,Z 471.893,A -85,B 0,C 180,E1 -461.323,E2 -461.323} C_VEL
LIN {X 0,Y 608.507,Z 459.537,A -85,B 0,C 180,E1 -461.639,E2 -461.639} C_VEL
LIN {X 0,Y 608.531,Z 443.772,A -85,B 0,C 180,E1 -461.871,E2 -461.871} C_VEL
LIN {X 0,Y 608.508,Z 347.183,A -85,B 0,C 180,E1 -463.015,E2 -463.015} C_VEL
LIN {X 0,Y 608.454,Z 346.131,A -85,B 0,C 180,E1 -463.101,E2 -463.101} C_VEL
LIN {X 0,Y 608.467,Z 327.361,A -85,B 0,C 180,E1 -465.577,E2 -465.577} C_VEL
LIN {X 0,Y 608.508,Z 307.945,A -85,B 0,C 180,E1 -468.17,E2 -468.17} C_VEL
LIN {X 0,Y 608.553,Z 287.233,A -85,B 0,C 180,E1 -470.977,E2 -470.977} C_VEL
LIN {X 0,Y 608.46,Z 274.688,A -85,B 0,C 180,E1 -472.714,E2 -472.714} C_VEL
LIN {X 0,Y 608.442,Z 274.689,A -85,B 0,C 180,E1 -475.301,E2 -475.301} C_VEL
LIN {X 0,Y 608.445,Z 274.69,A -85,B 0,C 180,E1 -477.518,E2 -477.518} C_VEL
LIN {X 0,Y 608.464,Z 274.694,A -85,B 0,C 180,E1 -479.971,E2 -479.971} C_VEL
LIN {X 0,Y 608.453,Z 274.687,A -85,B 0,C 180,E1 -482.879,E2 -482.879} C_VEL
LIN {X 0,Y 608.433,Z 274.689,A -85,B 0,C 180,E1 -485.278,E2 -485.278} C_VEL
LIN {X 0,Y 608.466,Z 274.687,A -85,B 0,C 180,E1 -487.746,E2 -487.746} C_VEL
LIN {X 0,Y 608.446,Z 274.698,A -85,B 0,C 180,E1 -490.328,E2 -490.328} C_VEL
LIN {X 0,Y 608.472,Z 274.684,A -85,B 0,C 180,E1 -493.309,E2 -493.309} C_VEL
LIN {X 0,Y 608.462,Z 274.69,A -85,B 0,C 180,E1 -496.13,E2 -496.13} C_VEL
LIN {X 0,Y 608.451,Z 274.694,A -85,B 0,C 180,E1 -498.823,E2 -498.823} C_VEL
LIN {X 0,Y 608.462,Z 274.686,A -85,B 0,C 180,E1 -501.411,E2 -501.411} C_VEL
LIN {X 0,Y 608.472,Z 274.684,A -85,B 0,C 180,E1 -503.95,E2 -503.95} C_VEL
LIN {X 0,Y 608.461,Z 274.689,A -85,B 0,C 180,E1 -506.329,E2 -506.329} C_VEL
LIN {X 0,Y 608.474,Z 274.693,A -85,B 0,C 180,E1 -508.727,E2 -508.727} C_VEL
LIN {X 0,Y 608.46,Z 274.689,A -85,B 0,C 180,E1 -511.381,E2 -511.381} C_VEL
LIN {X 0,Y 608.44,Z 274.688,A -85,B 0,C 180,E1 -513.964,E2 -513.964} C_VEL
LIN {X 0,Y 608.461,Z 274.685,A -85,B 0,C 180,E1 -516.155,E2 -516.155} C_VEL
LIN {X 0,Y 608.454,Z 274.695,A -85,B 0,C 180,E1 -519.018,E2 -519.018} C_VEL
LIN {X 0,Y 608.437,Z 274.69,A -85,B 0,C 180,E1 -521.828,E2 -521.828} C_VEL
LIN {X 0,Y 608.466,Z 274.686,A -85,B 0,C 180,E1 -524.594,E2 -524.594} C_VEL
LIN {X 0,Y 608.476,Z 274.694,A -85,B 0,C 180,E1 -527.323,E2 -527.323} C_VEL
LIN {X 0,Y 608.439,Z 274.69,A -85,B 0,C 180,E1 -530.023,E2 -530.023} C_VEL
LIN {X 0,Y 608.478,Z 274.684,A -85,B 0,C 180,E1 -532.701,E2 -532.701} C_VEL
LIN {X 0,Y 608.455,Z 274.693,A -85,B 0,C 180,E1 -535.362,E2 -535.362} C_VEL
LIN {X 0,Y 608.438,Z 274.693,A -85,B 0,C 180,E1 -538.014,E2 -538.014} C_VEL
LIN {X 0,Y 608.46,Z 274.685,A -85,B 0,C 180,E1 -540.662,E2 -540.662} C_VEL
LIN {X 0,Y 608.483,Z 274.686,A -85,B 0,C 180,E1 -543.311,E2 -543.311} C_VEL
LIN {X 0,Y 608.467,Z 274.695,A -85,B 0,C 180,E1 -545.967,E2 -545.967} C_VEL
LIN {X 0,Y 608.434,Z 274.69,A -85,B 0,C 180,E1 -548.637,E2 -548.637} C_VEL
LIN {X 0,Y 608.461,Z 274.688,A -85,B 0,C 180,E1 -549.441,E2 -549.441} C_VEL
LIN {X 0,Y 607.78,Z 274.782,A -85,B 0,C 180,E1 -549.993,E2 -549.993} C_VEL
LIN {X 0,Y 604.927,Z 275.141,A -85,B 0,C 180,E1 -550.89,E2 -550.89} C_VEL
LIN {X 0,Y 602.523,Z 275.439,A -85,B 0,C 180,E1 -551.612,E2 -551.612} C_VEL
LIN {X 0,Y 601.487,Z 275.564,A -85,B 0,C 180,E1 -552.168,E2 -552.168} C_VEL
LIN {X 0,Y 601.399,Z 275.571,A -85,B 0,C 180,E1 -552.357,E2 -552.357} C_VEL
LIN {X 0,Y 601.396,Z 275.566,A -85,B 0,C 180,E1 -554.898,E2 -554.898} C_VEL
LIN {X 0,Y 601.402,Z 275.565,A -85,B 0,C 180,E1 -556.987,E2 -556.987} C_VEL
LIN {X 0,Y 601.399,Z 275.569,A -85,B 0,C 180,E1 -559.81,E2 -559.81} C_VEL
LIN {X 0,Y 601.405,Z 275.569,A -85,B 0,C 180,E1 -562.684,E2 -562.684} C_VEL
LIN {X 0,Y 601.387,Z 275.57,A -85,B 0,C 180,E1 -564.88,E2 -564.88} C_VEL
LIN {X 0,Y 601.383,Z 275.567,A -85,B 0,C 180,E1 -567.358,E2 -567.358} C_VEL
LIN {X 0,Y 601.394,Z 275.566,A -85,B 0,C 180,E1 -569.395,E2 -569.395} C_VEL
LIN {X 0,Y 601.394,Z 275.566,A -85,B 0,C 180,E1 -571.728,E2 -571.728} C_VEL
LIN {X 0,Y 601.418,Z 275.565,A -85,B 0,C 180,E1 -574.119,E2 -574.119} C_VEL
LIN {X 0,Y 601.425,Z 275.563,A -85,B 0,C 180,E1 -577.382,E2 -577.382} C_VEL
LIN {X 0,Y 601.393,Z 275.566,A -85,B 0,C 180,E1 -579.997,E2 -579.997} C_VEL
LIN {X 0,Y 601.41,Z 275.571,A -85,B 0,C 180,E1 -582.671,E2 -582.671} C_VEL
LIN {X 0,Y 601.397,Z 275.568,A -85,B 0,C 180,E1 -585.48,E2 -585.48} C_VEL
LIN {X 0,Y 601.417,Z 275.564,A -85,B 0,C 180,E1 -588.408,E2 -588.408} C_VEL
LIN {X 0,Y 601.399,Z 275.569,A -85,B 0,C 180,E1 -591.534,E2 -591.534} C_VEL
LIN {X 0,Y 601.387,Z 275.569,A -85,B 0,C 180,E1 -593.742,E2 -593.742} C_VEL
LIN {X 0,Y 601.402,Z 275.565,A -85,B 0,C 180,E1 -596.07,E2 -596.07} C_VEL
LIN {X 0,Y 601.411,Z 275.564,A -85,B 0,C 180,E1 -598.548,E2 -598.548} C_VEL
LIN {X 0,Y 601.427,Z 275.573,A -85,B 0,C 180,E1 -601.374,E2 -601.374} C_VEL
LIN {X 0,Y 601.376,Z 275.569,A -85,B 0,C 180,E1 -604.141,E2 -604.141} C_VEL
LIN {X 0,Y 601.37,Z 275.569,A -85,B 0,C 180,E1 -606.588,E2 -606.588} C_VEL
LIN {X 0,Y 601.43,Z 275.57,A -85,B 0,C 180,E1 -609.479,E2 -609.479} C_VEL
LIN {X 0,Y 601.364,Z 275.571,A -85,B 0,C 180,E1 -612.311,E2 -612.311} C_VEL
LIN {X 0,Y 601.375,Z 275.569,A -85,B 0,C 180,E1 -614.408,E2 -614.408} C_VEL
LIN {X 0,Y 601.374,Z 275.569,A -85,B 0,C 180,E1 -616.484,E2 -616.484} C_VEL
LIN {X 0,Y 601.377,Z 275.569,A -85,B 0,C 180,E1 -619.224,E2 -619.224} C_VEL
LIN {X 0,Y 601.41,Z 275.575,A -85,B 0,C 180,E1 -621.939,E2 -621.939} C_VEL
LIN {X 0,Y 601.383,Z 275.569,A -85,B 0,C 180,E1 -624.636,E2 -624.636} C_VEL
LIN {X 0,Y 601.397,Z 275.566,A -85,B 0,C 180,E1 -627.321,E2 -627.321} C_VEL
LIN {X 0,Y 601.445,Z 275.567,A -85,B 0,C 180,E1 -630,E2 -630} C_VEL
LIN {X 0,Y 601.406,Z 275.568,A -85,B 0,C 180,E1 -632.68,E2 -632.68} C_VEL
LIN {X 0,Y 601.372,Z 275.568,A -85,B 0,C 180,E1 -635.365,E2 -635.365} C_VEL
LIN {X 0,Y 601.391,Z 275.571,A -85,B 0,C 180,E1 -638.062,E2 -638.062} C_VEL
LIN {X 0,Y 601.363,Z 275.572,A -85,B 0,C 180,E1 -640.979,E2 -640.979} C_VEL
LIN {X 0,Y 601.359,Z 275.57,A -85,B 0,C 180,E1 -643.518,E2 -643.518} C_VEL
LIN {X 0,Y 601.414,Z 275.569,A -85,B 0,C 180,E1 -646.288,E2 -646.288} C_VEL
LIN {X 0,Y 601.398,Z 275.569,A -85,B 0,C 180,E1 -649.1,E2 -649.1} C_VEL
LIN {X 0,Y 601.369,Z 275.572,A -85,B 0,C 180,E1 -651.241,E2 -651.241} C_VEL
LIN {X 0,Y 601.353,Z 275.573,A -85,B 0,C 180,E1 -653.413,E2 -653.413} C_VEL
LIN {X 0,Y 601.341,Z 275.573,A -85,B 0,C 180,E1 -655.852,E2 -655.852} C_VEL
LIN {X 0,Y 601.371,Z 275.626,A -85,B 0,C 180,E1 -658.249,E2 -658.249} C_VEL
LIN {X 0,Y 601.45,Z 288.889,A -85,B 0,C 180,E1 -660.551,E2 -660.551} C_VEL
LIN {X 0,Y 601.408,Z 305.049,A -85,B 0,C 180,E1 -663.315,E2 -663.315} C_VEL
LIN {X 0,Y 601.399,Z 308.442,A -85,B 0,C 180,E1 -663.888,E2 -663.888} C_VEL
LIN {X 0,Y 601.658,Z 317.581,A -85,B 0,C 180,E1 -664.004,E2 -664.004} C_VEL
LIN {X 0,Y 601.605,Z 415.09,A -85,B 0,C 180,E1 -665.187,E2 -665.187} C_VEL
LIN {X 0,Y 601.539,Z 429.239,A -85,B 0,C 180,E1 -665.511,E2 -665.511} C_VEL
LIN {X 0,Y 601.533,Z 441.307,A -85,B 0,C 180,E1 -665.924,E2 -665.924} C_VEL
LIN {X 0,Y 601.509,Z 453.277,A -85,B 0,C 180,E1 -666.475,E2 -666.475} C_VEL
LIN {X 0,Y 601.477,Z 465.252,A -85,B 0,C 180,E1 -667.191,E2 -667.191} C_VEL
LIN {X 0,Y 601.44,Z 475.392,A -85,B 0,C 180,E1 -667.948,E2 -667.948} C_VEL
LIN {X 0,Y 601.412,Z 484.257,A -85,B 0,C 180,E1 -668.769,E2 -668.769} C_VEL
LIN {X 0,Y 601.396,Z 491.28,A -85,B 0,C 180,E1 -669.53,E2 -669.53} C_VEL
LIN {X 0,Y 601.353,Z 499.031,A -85,B 0,C 180,E1 -670.566,E2 -670.566} C_VEL
LIN {X 0,Y 601.367,Z 505.163,A -85,B 0,C 180,E1 -671.586,E2 -671.586} C_VEL
LIN {X 0,Y 601.352,Z 510.311,A -85,B 0,C 180,E1 -672.676,E2 -672.676} C_VEL
LIN {X 0,Y 601.348,Z 513.633,A -85,B 0,C 180,E1 -673.594,E2 -673.594} C_VEL
LIN {X 0,Y 601.339,Z 516.166,A -85,B 0,C 180,E1 -674.526,E2 -674.526} C_VEL
LIN {X 0,Y 601.339,Z 517.898,A -85,B 0,C 180,E1 -675.473,E2 -675.473} C_VEL
LIN {X 0,Y 601.347,Z 518.825,A -85,B 0,C 180,E1 -676.436,E2 -676.436} C_VEL
LIN {X 0,Y 601.345,Z 518.92,A -85,B 0,C 180,E1 -677.416,E2 -677.416} C_VEL
LIN {X 0,Y 601.326,Z 518.145,A -85,B 0,C 180,E1 -678.418,E2 -678.418} C_VEL
LIN {X 0,Y 601.323,Z 516.436,A -85,B 0,C 180,E1 -679.437,E2 -679.437} C_VEL
LIN {X 0,Y 601.325,Z 513.692,A -85,B 0,C 180,E1 -680.478,E2 -680.478} C_VEL
LIN {X 0,Y 601.327,Z 509.773,A -85,B 0,C 180,E1 -681.542,E2 -681.542} C_VEL
LIN {X 0,Y 601.366,Z 504.5,A -85,B 0,C 180,E1 -682.627,E2 -682.627} C_VEL
LIN {X 0,Y 601.376,Z 497.567,A -85,B 0,C 180,E1 -683.743,E2 -683.743} C_VEL
LIN {X 0,Y 601.396,Z 489.491,A -85,B 0,C 180,E1 -684.767,E2 -684.767} C_VEL
LIN {X 0,Y 601.435,Z 479.539,A -85,B 0,C 180,E1 -685.78,E2 -685.78} C_VEL
LIN {X 0,Y 601.471,Z 469.645,A -85,B 0,C 180,E1 -686.589,E2 -686.589} C_VEL
LIN {X 0,Y 601.47,Z 458.196,A -85,B 0,C 180,E1 -687.343,E2 -687.343} C_VEL
LIN {X 0,Y 601.542,Z 446.71,A -85,B 0,C 180,E1 -687.936,E2 -687.936} C_VEL
LIN {X 0,Y 601.532,Z 434.838,A -85,B 0,C 180,E1 -688.403,E2 -688.403} C_VEL
LIN {X 0,Y 601.539,Z 422.391,A -85,B 0,C 180,E1 -688.756,E2 -688.756} C_VEL
LIN {X 0,Y 601.555,Z 409.727,A -85,B 0,C 180,E1 -688.983,E2 -688.983} C_VEL
LIN {X 0,Y 601.59,Z 309.663,A -85,B 0,C 180,E1 -690.183,E2 -690.183} C_VEL
LIN {X 0,Y 601.428,Z 308.302,A -85,B 0,C 180,E1 -690.222,E2 -690.222} C_VEL
LIN {X 0,Y 601.443,Z 292.675,A -85,B 0,C 180,E1 -692.888,E2 -692.888} C_VEL
LIN {X 0,Y 601.477,Z 276.418,A -85,B 0,C 180,E1 -695.699,E2 -695.699} C_VEL
LIN {X 0,Y 601.448,Z 275.562,A -85,B 0,C 180,E1 -695.859,E2 -695.859} C_VEL
LIN {X 0,Y 601.407,Z 275.568,A -85,B 0,C 180,E1 -698.76,E2 -698.76} C_VEL
LIN {X 0,Y 601.418,Z 275.569,A -85,B 0,C 180,E1 -701.608,E2 -701.608} C_VEL
LIN {X 0,Y 601.409,Z 275.564,A -85,B 0,C 180,E1 -704.408,E2 -704.408} C_VEL
LIN {X 0,Y 601.419,Z 275.568,A -85,B 0,C 180,E1 -707.172,E2 -707.172} C_VEL
LIN {X 0,Y 601.426,Z 275.568,A -85,B 0,C 180,E1 -709.905,E2 -709.905} C_VEL
LIN {X 0,Y 601.44,Z 275.56,A -85,B 0,C 180,E1 -712.615,E2 -712.615} C_VEL
LIN {X 0,Y 601.418,Z 275.566,A -85,B 0,C 180,E1 -715.308,E2 -715.308} C_VEL
LIN {X 0,Y 601.424,Z 275.571,A -85,B 0,C 180,E1 -717.991,E2 -717.991} C_VEL
LIN {X 0,Y 601.441,Z 275.561,A -85,B 0,C 180,E1 -720.669,E2 -720.669} C_VEL
LIN {X 0,Y 601.432,Z 275.562,A -85,B 0,C 180,E1 -723.349,E2 -723.349} C_VEL
LIN {X 0,Y 601.409,Z 275.574,A -85,B 0,C 180,E1 -726.037,E2 -726.037} C_VEL
LIN {X 0,Y 601.411,Z 275.566,A -85,B 0,C 180,E1 -728.738,E2 -728.738} C_VEL
LIN {X 0,Y 601.434,Z 275.561,A -85,B 0,C 180,E1 -731.458,E2 -731.458} C_VEL
LIN {X 0,Y 601.421,Z 275.57,A -85,B 0,C 180,E1 -734.205,E2 -734.205} C_VEL
LIN {X 0,Y 601.42,Z 275.565,A -85,B 0,C 180,E1 -736.986,E2 -736.986} C_VEL
LIN {X 0,Y 601.402,Z 275.565,A -85,B 0,C 180,E1 -739.81,E2 -739.81} C_VEL
LIN {X 0,Y 601.417,Z 275.573,A -85,B 0,C 180,E1 -742.606,E2 -742.606} C_VEL
LIN {X 0,Y 601.396,Z 275.574,A -85,B 0,C 180,E1 -744.879,E2 -744.879} C_VEL
LIN {X 0,Y 601.41,Z 275.566,A -85,B 0,C 180,E1 -747.361,E2 -747.361} C_VEL
LIN {X 0,Y 601.43,Z 275.562,A -85,B 0,C 180,E1 -750.164,E2 -750.164} C_VEL
LIN {X 0,Y 601.417,Z 275.569,A -85,B 0,C 180,E1 -752.715,E2 -752.715} C_VEL
LIN {X 0,Y 601.39,Z 275.577,A -85,B 0,C 180,E1 -755.111,E2 -755.111} C_VEL
LIN {X 0,Y 601.436,Z 275.567,A -85,B 0,C 180,E1 -757.419,E2 -757.419} C_VEL
LIN {X 0,Y 601.402,Z 275.565,A -85,B 0,C 180,E1 -759.996,E2 -759.996} C_VEL
LIN {X 0,Y 601.413,Z 275.565,A -85,B 0,C 180,E1 -762.67,E2 -762.67} C_VEL
LIN {X 0,Y 601.4,Z 275.575,A -85,B 0,C 180,E1 -765.479,E2 -765.479} C_VEL
LIN {X 0,Y 601.423,Z 275.562,A -85,B 0,C 180,E1 -768.407,E2 -768.407} C_VEL
LIN {X 0,Y 601.427,Z 275.572,A -85,B 0,C 180,E1 -771.53,E2 -771.53} C_VEL
LIN {X 0,Y 601.384,Z 275.57,A -85,B 0,C 180,E1 -774.245,E2 -774.245} C_VEL
LIN {X 0,Y 601.416,Z 275.563,A -85,B 0,C 180,E1 -776.686,E2 -776.686} C_VEL
LIN {X 0,Y 601.417,Z 275.564,A -85,B 0,C 180,E1 -779.058,E2 -779.058} C_VEL
LIN {X 0,Y 601.43,Z 275.564,A -85,B 0,C 180,E1 -781.373,E2 -781.373} C_VEL
LIN {X 0,Y 601.399,Z 275.571,A -85,B 0,C 180,E1 -783.636,E2 -783.636} C_VEL
LIN {X 0,Y 601.418,Z 275.569,A -85,B 0,C 180,E1 -786.589,E2 -786.589} C_VEL
LIN {X 0,Y 601.421,Z 275.577,A -85,B 0,C 180,E1 -787.136,E2 -787.136} C_VEL
LIN {X 0,Y 601.673,Z 282.049,A -85,B 0,C 180,E1 -788.051,E2 -788.051} C_VEL
LIN {X 0,Y 601.602,Z 302.761,A -85,B 0,C 180,E1 -790.907,E2 -790.907} C_VEL
LIN {X 0,Y 601.525,Z 323.472,A -85,B 0,C 180,E1 -793.715,E2 -793.715} C_VEL
LIN {X 0,Y 601.468,Z 344.183,A -85,B 0,C 180,E1 -796.485,E2 -796.485} C_VEL
LIN {X 0,Y 601.426,Z 346.611,A -85,B 0,C 180,E1 -796.807,E2 -796.807} C_VEL
LIN {X 0,Y 601.667,Z 350.694,A -85,B 0,C 180,E1 -796.876,E2 -796.876} C_VEL
LIN {X 0,Y 601.594,Z 454.93,A -85,B 0,C 180,E1 -798.139,E2 -798.139} C_VEL
LIN {X 0,Y 601.556,Z 468.206,A -85,B 0,C 180,E1 -798.437,E2 -798.437} C_VEL
LIN {X 0,Y 601.542,Z 479.912,A -85,B 0,C 180,E1 -798.826,E2 -798.826} C_VEL
LIN {X 0,Y 601.521,Z 492.627,A -85,B 0,C 180,E1 -799.396,E2 -799.396} C_VEL
LIN {X 0,Y 601.472,Z 504.194,A -85,B 0,C 180,E1 -800.075,E2 -800.075} C_VEL
LIN {X 0,Y 601.444,Z 514.591,A -85,B 0,C 180,E1 -800.839,E2 -800.839} C_VEL
LIN {X 0,Y 601.405,Z 523.012,A -85,B 0,C 180,E1 -801.6,E2 -801.6} C_VEL
LIN {X 0,Y 601.418,Z 530.957,A -85,B 0,C 180,E1 -802.445,E2 -802.445} C_VEL
LIN {X 0,Y 601.366,Z 538.247,A -85,B 0,C 180,E1 -803.401,E2 -803.401} C_VEL
LIN {X 0,Y 601.372,Z 543.864,A -85,B 0,C 180,E1 -804.299,E2 -804.299} C_VEL
LIN {X 0,Y 601.336,Z 548.948,A -85,B 0,C 180,E1 -805.307,E2 -805.307} C_VEL
LIN {X 0,Y 601.367,Z 552.895,A -85,B 0,C 180,E1 -806.314,E2 -806.314} C_VEL
LIN {X 0,Y 601.325,Z 555.808,A -85,B 0,C 180,E1 -807.32,E2 -807.32} C_VEL
LIN {X 0,Y 601.341,Z 557.201,A -85,B 0,C 180,E1 -807.99,E2 -807.99} C_VEL
LIN {X 0,Y 601.339,Z 558.784,A -85,B 0,C 180,E1 -809.33,E2 -809.33} C_VEL
LIN {X 0,Y 601.335,Z 559,A -85,B 0,C 180,E1 -810,E2 -810} C_VEL
LIN {X 0,Y 601.347,Z 558.185,A -85,B 0,C 180,E1 -811.339,E2 -811.339} C_VEL
LIN {X 0,Y 601.341,Z 557.203,A -85,B 0,C 180,E1 -812.009,E2 -812.009} C_VEL
LIN {X 0,Y 601.325,Z 555.81,A -85,B 0,C 180,E1 -812.679,E2 -812.679} C_VEL
LIN {X 0,Y 601.367,Z 552.897,A -85,B 0,C 180,E1 -813.685,E2 -813.685} C_VEL
LIN {X 0,Y 601.336,Z 548.952,A -85,B 0,C 180,E1 -814.692,E2 -814.692} C_VEL
LIN {X 0,Y 601.372,Z 542.88,A -85,B 0,C 180,E1 -815.869,E2 -815.869} C_VEL
LIN {X 0,Y 601.381,Z 536.239,A -85,B 0,C 180,E1 -816.879,E2 -816.879} C_VEL
LIN {X 0,Y 601.4,Z 527.993,A -85,B 0,C 180,E1 -817.892,E2 -817.892} C_VEL
LIN {X 0,Y 601.434,Z 517.604,A -85,B 0,C 180,E1 -818.907,E2 -818.907} C_VEL
LIN {X 0,Y 601.46,Z 506.754,A -85,B 0,C 180,E1 -819.754,E2 -819.754} C_VEL
LIN {X 0,Y 601.494,Z 495.784,A -85,B 0,C 180,E1 -820.434,E2 -820.434} C_VEL
LIN {X 0,Y 601.548,Z 483.683,A -85,B 0,C 180,E1 -821.022,E2 -821.022} C_VEL
LIN {X 0,Y 601.53,Z 471.892,A -85,B 0,C 180,E1 -821.456,E2 -821.456} C_VEL
LIN {X 0,Y 601.577,Z 459.536,A -85,B 0,C 180,E1 -821.775,E2 -821.775} C_VEL
LIN {X 0,Y 601.607,Z 443.772,A -85,B 0,C 180,E1 -822.01,E2 -822.01} C_VEL
LIN {X 0,Y 601.478,Z 347.183,A -85,B 0,C 180,E1 -823.17,E2 -823.17} C_VEL
LIN {X 0,Y 601.461,Z 346.131,A -85,B 0,C 180,E1 -823.256,E2 -823.256} C_VEL
LIN {X 0,Y 601.466,Z 326.067,A -85,B 0,C 180,E1 -825.937,E2 -825.937} C_VEL
LIN {X 0,Y 601.565,Z 306.198,A -85,B 0,C 180,E1 -828.625,E2 -828.625} C_VEL
LIN {X 0,Y 601.654,Z 284.644,A -85,B 0,C 180,E1 -831.589,E2 -831.589} C_VEL
LIN {X 0,Y 601.673,Z 276.878,A -85,B 0,C 180,E1 -832.672,E2 -832.672} C_VEL
LIN {X 0,Y 601.416,Z 275.567,A -85,B 0,C 180,E1 -832.886,E2 -832.886} C_VEL
LIN {X 0,Y 601.398,Z 275.566,A -85,B 0,C 180,E1 -834.878,E2 -834.878} C_VEL
LIN {X 0,Y 601.417,Z 275.572,A -85,B 0,C 180,E1 -837.867,E2 -837.867} C_VEL
LIN {X 0,Y 601.428,Z 275.572,A -85,B 0,C 180,E1 -840.163,E2 -840.163} C_VEL
LIN {X 0,Y 601.418,Z 275.565,A -85,B 0,C 180,E1 -842.715,E2 -842.715} C_VEL
LIN {X 0,Y 601.39,Z 275.566,A -85,B 0,C 180,E1 -845.111,E2 -845.111} C_VEL
LIN {X 0,Y 601.434,Z 275.561,A -85,B 0,C 180,E1 -847.418,E2 -847.418} C_VEL
LIN {X 0,Y 601.398,Z 275.57,A -85,B 0,C 180,E1 -849.995,E2 -849.995} C_VEL
LIN {X 0,Y 601.41,Z 275.571,A -85,B 0,C 180,E1 -852.67,E2 -852.67} C_VEL
LIN {X 0,Y 601.423,Z 275.562,A -85,B 0,C 180,E1 -855.482,E2 -855.482} C_VEL
LIN {X 0,Y 601.423,Z 275.57,A -85,B 0,C 180,E1 -858.406,E2 -858.406} C_VEL
LIN {X 0,Y 601.429,Z 275.569,A -85,B 0,C 180,E1 -860.875,E2 -860.875} C_VEL
LIN {X 0,Y 601.438,Z 275.56,A -85,B 0,C 180,E1 -863.734,E2 -863.734} C_VEL
LIN {X 0,Y 601.423,Z 275.571,A -85,B 0,C 180,E1 -866.686,E2 -866.686} C_VEL
LIN {X 0,Y 601.427,Z 275.57,A -85,B 0,C 180,E1 -869.058,E2 -869.058} C_VEL
LIN {X 0,Y 601.42,Z 275.566,A -85,B 0,C 180,E1 -871.373,E2 -871.373} C_VEL
LIN {X 0,Y 601.399,Z 275.567,A -85,B 0,C 180,E1 -873.636,E2 -873.636} C_VEL
LIN {X 0,Y 601.417,Z 275.566,A -85,B 0,C 180,E1 -876.59,E2 -876.59} C_VEL
LIN {X 0,Y 601.423,Z 275.568,A -85,B 0,C 180,E1 -879.478,E2 -879.478} C_VEL
LIN {X 0,Y 601.389,Z 275.566,A -85,B 0,C 180,E1 -882.311,E2 -882.311} C_VEL
LIN {X 0,Y 601.407,Z 275.564,A -85,B 0,C 180,E1 -884.409,E2 -884.409} C_VEL
LIN {X 0,Y 601.42,Z 275.57,A -85,B 0,C 180,E1 -887.172,E2 -887.172} C_VEL
LIN {X 0,Y 601.42,Z 275.566,A -85,B 0,C 180,E1 -889.905,E2 -889.905} C_VEL
LIN {X 0,Y 601.447,Z 275.559,A -85,B 0,C 180,E1 -892.615,E2 -892.615} C_VEL
LIN {X 0,Y 601.423,Z 275.568,A -85,B 0,C 180,E1 -895.308,E2 -895.308} C_VEL
LIN {X 0,Y 601.41,Z 275.569,A -85,B 0,C 180,E1 -897.991,E2 -897.991} C_VEL
LIN {X 0,Y 601.433,Z 275.561,A -85,B 0,C 180,E1 -900.67,E2 -900.67} C_VEL
LIN {X 0,Y 601.434,Z 275.564,A -85,B 0,C 180,E1 -903.35,E2 -903.35} C_VEL
LIN {X 0,Y 601.414,Z 275.572,A -85,B 0,C 180,E1 -906.037,E2 -906.037} C_VEL
LIN {X 0,Y 601.435,Z 275.57,A -85,B 0,C 180,E1 -908.061,E2 -908.061} C_VEL
LIN {X 0,Y 601.408,Z 275.564,A -85,B 0,C 180,E1 -911.008,E2 -911.008} C_VEL
LIN {X 0,Y 601.399,Z 275.571,A -85,B 0,C 180,E1 -912.357,E2 -912.357} C_VEL
LIN {X 0,Y 600.724,Z 275.651,A -85,B 0,C 180,E1 -912.916,E2 -912.916} C_VEL
LIN {X 0,Y 597.864,Z 276.012,A -85,B 0,C 180,E1 -913.824,E2 -913.824} C_VEL
LIN {X 0,Y 595.456,Z 276.309,A -85,B 0,C 180,E1 -914.554,E2 -914.554} C_VEL
LIN {X 0,Y 594.425,Z 276.434,A -85,B 0,C 180,E1 -915.118,E2 -915.118} C_VEL
LIN {X 0,Y 594.343,Z 276.444,A -85,B 0,C 180,E1 -915.308,E2 -915.308} C_VEL
LIN {X 0,Y 594.345,Z 276.45,A -85,B 0,C 180,E1 -917.906,E2 -917.906} C_VEL
LIN {X 0,Y 594.39,Z 276.441,A -85,B 0,C 180,E1 -920.776,E2 -920.776} C_VEL
LIN {X 0,Y 594.374,Z 276.442,A -85,B 0,C 180,E1 -923.705,E2 -923.705} C_VEL
LIN {X 0,Y 594.355,Z 276.449,A -85,B 0,C 180,E1 -926.701,E2 -926.701} C_VEL
LIN {X 0,Y 594.372,Z 276.444,A -85,B 0,C 180,E1 -928.999,E2 -928.999} C_VEL
LIN {X 0,Y 594.369,Z 276.441,A -85,B 0,C 180,E1 -931.643,E2 -931.643} C_VEL
LIN {X 0,Y 594.373,Z 276.45,A -85,B 0,C 180,E1 -934.581,E2 -934.581} C_VEL
LIN {X 0,Y 594.381,Z 276.439,A -85,B 0,C 180,E1 -937.609,E2 -937.609} C_VEL
LIN {X 0,Y 594.361,Z 276.448,A -85,B 0,C 180,E1 -940.568,E2 -940.568} C_VEL
LIN {X 0,Y 594.349,Z 276.448,A -85,B 0,C 180,E1 -943.302,E2 -943.302} C_VEL
LIN {X 0,Y 594.357,Z 276.443,A -85,B 0,C 180,E1 -946.162,E2 -946.162} C_VEL
LIN {X 0,Y 594.374,Z 276.449,A -85,B 0,C 180,E1 -949.179,E2 -949.179} C_VEL
LIN {X 0,Y 594.367,Z 276.441,A -85,B 0,C 180,E1 -952.059,E2 -952.059} C_VEL
LIN {X 0,Y 594.35,Z 276.446,A -85,B 0,C 180,E1 -954.677,E2 -954.677} C_VEL
LIN {X 0,Y 594.374,Z 276.448,A -85,B 0,C 180,E1 -957.09,E2 -957.09} C_VEL
LIN {X 0,Y 594.348,Z 276.449,A -85,B 0,C 180,E1 -959.679,E2 -959.679} C_VEL
LIN {X 0,Y 594.337,Z 276.45,A -85,B 0,C 180,E1 -961.772,E2 -961.772} C_VEL
LIN {X 0,Y 594.34,Z 276.446,A -85,B 0,C 180,E1 -964.055,E2 -964.055} C_VEL
LIN {X 0,Y 594.353,Z 276.443,A -85,B 0,C 180,E1 -966.295,E2 -966.295} C_VEL
LIN {X 0,Y 594.406,Z 276.441,A -85,B 0,C 180,E1 -969.225,E2 -969.225} C_VEL
LIN {X 0,Y 594.326,Z 276.45,A -85,B 0,C 180,E1 -972.095,E2 -972.095} C_VEL
LIN {X 0,Y 594.337,Z 276.448,A -85,B 0,C 180,E1 -974.219,E2 -974.219} C_VEL
LIN {X 0,Y 594.349,Z 276.446,A -85,B 0,C 180,E1 -976.321,E2 -976.321} C_VEL
LIN {X 0,Y 594.335,Z 276.445,A -85,B 0,C 180,E1 -978.957,E2 -978.957} C_VEL
LIN {X 0,Y 594.36,Z 276.451,A -85,B 0,C 180,E1 -981.843,E2 -981.843} C_VEL
LIN {X 0,Y 594.353,Z 276.445,A -85,B 0,C 180,E1 -984.572,E2 -984.572} C_VEL
LIN {X 0,Y 594.365,Z 276.442,A -85,B 0,C 180,E1 -987.289,E2 -987.289} C_VEL
LIN {X 0,Y 594.414,Z 276.443,A -85,B 0,C 180,E1 -990,E2 -990} C_VEL
LIN {X 0,Y 594.372,Z 276.444,A -85,B 0,C 180,E1 -992.711,E2 -992.711} C_VEL
LIN {X 0,Y 594.342,Z 276.444,A -85,B 0,C 180,E1 -995.429,E2 -995.429} C_VEL
LIN {X 0,Y 594.346,Z 276.451,A -85,B 0,C 180,E1 -998.158,E2 -998.158} C_VEL
LIN {X 0,Y 594.336,Z 276.447,A -85,B 0,C 180,E1 -1001.044,E2 -1001.044} C_VEL
LIN {X 0,Y 594.331,Z 276.446,A -85,B 0,C 180,E1 -1003.68,E2 -1003.68} C_VEL
LIN {X 0,Y 594.365,Z 276.451,A -85,B 0,C 180,E1 -1006.708,E2 -1006.708} C_VEL
LIN {X 0,Y 594.345,Z 276.445,A -85,B 0,C 180,E1 -1009.335,E2 -1009.335} C_VEL
LIN {X 0,Y 594.324,Z 276.447,A -85,B 0,C 180,E1 -1011.505,E2 -1011.505} C_VEL
LIN {X 0,Y 594.314,Z 276.448,A -85,B 0,C 180,E1 -1013.707,E2 -1013.707} C_VEL
LIN {X 0,Y 594.34,Z 276.453,A -85,B 0,C 180,E1 -1016.702,E2 -1016.702} C_VEL
LIN {X 0,Y 594.317,Z 276.556,A -85,B 0,C 180,E1 -1018.182,E2 -1018.182} C_VEL
LIN {X 0,Y 594.403,Z 285.601,A -85,B 0,C 180,E1 -1019.775,E2 -1019.775} C_VEL
LIN {X 0,Y 594.425,Z 301.428,A -85,B 0,C 180,E1 -1022.526,E2 -1022.526} C_VEL
LIN {X 0,Y 594.357,Z 308.323,A -85,B 0,C 180,E1 -1023.712,E2 -1023.712} C_VEL
LIN {X 0,Y 594.763,Z 312.614,A -85,B 0,C 180,E1 -1023.79,E2 -1023.79} C_VEL
LIN {X 0,Y 594.67,Z 415.328,A -85,B 0,C 180,E1 -1025.051,E2 -1025.051} C_VEL
LIN {X 0,Y 594.601,Z 429.231,A -85,B 0,C 180,E1 -1025.374,E2 -1025.374} C_VEL
LIN {X 0,Y 594.572,Z 441.714,A -85,B 0,C 180,E1 -1025.81,E2 -1025.81} C_VEL
LIN {X 0,Y 594.52,Z 453.534,A -85,B 0,C 180,E1 -1026.364,E2 -1026.364} C_VEL
LIN {X 0,Y 594.462,Z 465.377,A -85,B 0,C 180,E1 -1027.081,E2 -1027.081} C_VEL
LIN {X 0,Y 594.403,Z 476.542,A -85,B 0,C 180,E1 -1027.94,E2 -1027.94} C_VEL
LIN {X 0,Y 594.347,Z 485.637,A -85,B 0,C 180,E1 -1028.808,E2 -1028.808} C_VEL
LIN {X 0,Y 594.308,Z 493.86,A -85,B 0,C 180,E1 -1029.766,E2 -1029.766} C_VEL
LIN {X 0,Y 594.268,Z 501.119,A -85,B 0,C 180,E1 -1030.809,E2 -1030.809} C_VEL
LIN {X 0,Y 594.266,Z 507.986,A -85,B 0,C 180,E1 -1032.086,E2 -1032.086} C_VEL
LIN {X 0,Y 594.255,Z 512.857,A -85,B 0,C 180,E1 -1033.31,E2 -1033.31} C_VEL
LIN {X 0,Y 594.24,Z 515.595,A -85,B 0,C 180,E1 -1034.25,E2 -1034.25} C_VEL
LIN {X 0,Y 594.234,Z 517.515,A -85,B 0,C 180,E1 -1035.204,E2 -1035.204} C_VEL
LIN {X 0,Y 594.24,Z 518.651,A -85,B 0,C 180,E1 -1036.174,E2 -1036.174} C_VEL
LIN {X 0,Y 594.25,Z 518.98,A -85,B 0,C 180,E1 -1037.16,E2 -1037.16} C_VEL
LIN {X 0,Y 594.221,Z 518.042,A -85,B 0,C 180,E1 -1038.522,E2 -1038.522} C_VEL
LIN {X 0,Y 594.244,Z 516.526,A -85,B 0,C 180,E1 -1039.422,E2 -1039.422} C_VEL
LIN {X 0,Y 594.23,Z 514.347,A -85,B 0,C 180,E1 -1040.307,E2 -1040.307} C_VEL
LIN {X 0,Y 594.248,Z 510.949,A -85,B 0,C 180,E1 -1041.312,E2 -1041.312} C_VEL
LIN {X 0,Y 594.261,Z 506.015,A -85,B 0,C 180,E1 -1042.408,E2 -1042.408} C_VEL
LIN {X 0,Y 594.313,Z 499.518,A -85,B 0,C 180,E1 -1043.526,E2 -1043.526} C_VEL
LIN {X 0,Y 594.318,Z 491.767,A -85,B 0,C 180,E1 -1044.588,E2 -1044.588} C_VEL
LIN {X 0,Y 594.372,Z 484.273,A -85,B 0,C 180,E1 -1045.419,E2 -1045.419} C_VEL
LIN {X 0,Y 594.406,Z 475.522,A -85,B 0,C 180,E1 -1046.24,E2 -1046.24} C_VEL
LIN {X 0,Y 594.446,Z 464.342,A -85,B 0,C 180,E1 -1047.079,E2 -1047.079} C_VEL
LIN {X 0,Y 594.507,Z 452.865,A -85,B 0,C 180,E1 -1047.761,E2 -1047.761} C_VEL
LIN {X 0,Y 594.564,Z 441.622,A -85,B 0,C 180,E1 -1048.284,E2 -1048.284} C_VEL
LIN {X 0,Y 594.58,Z 428.988,A -85,B 0,C 180,E1 -1048.724,E2 -1048.724} C_VEL
LIN {X 0,Y 594.631,Z 414.896,A -85,B 0,C 180,E1 -1049.048,E2 -1049.048} C_VEL
LIN {X 0,Y 594.629,Z 310.038,A -85,B 0,C 180,E1 -1050.335,E2 -1050.335} C_VEL
LIN {X 0,Y 594.395,Z 308.362,A -85,B 0,C 180,E1 -1050.371,E2 -1050.371} C_VEL
LIN {X 0,Y 594.434,Z 293.58,A -85,B 0,C 180,E1 -1052.923,E2 -1052.923} C_VEL
LIN {X 0,Y 594.475,Z 278.513,A -85,B 0,C 180,E1 -1055.557,E2 -1055.557} C_VEL
LIN {X 0,Y 594.405,Z 276.44,A -85,B 0,C 180,E1 -1055.949,E2 -1055.949} C_VEL
LIN {X 0,Y 594.404,Z 276.448,A -85,B 0,C 180,E1 -1059.224,E2 -1059.224} C_VEL
LIN {X 0,Y 594.35,Z 276.445,A -85,B 0,C 180,E1 -1062.095,E2 -1062.095} C_VEL
LIN {X 0,Y 594.362,Z 276.443,A -85,B 0,C 180,E1 -1064.219,E2 -1064.219} C_VEL
LIN {X 0,Y 594.378,Z 276.44,A -85,B 0,C 180,E1 -1066.321,E2 -1066.321} C_VEL
LIN {X 0,Y 594.377,Z 276.443,A -85,B 0,C 180,E1 -1069.094,E2 -1069.094} C_VEL
LIN {X 0,Y 594.381,Z 276.448,A -85,B 0,C 180,E1 -1071.843,E2 -1071.843} C_VEL
LIN {X 0,Y 594.392,Z 276.439,A -85,B 0,C 180,E1 -1074.572,E2 -1074.572} C_VEL
LIN {X 0,Y 594.404,Z 276.439,A -85,B 0,C 180,E1 -1077.289,E2 -1077.289} C_VEL
LIN {X 0,Y 594.414,Z 276.445,A -85,B 0,C 180,E1 -1080,E2 -1080} C_VEL
LIN {X 0,Y 594.398,Z 276.438,A -85,B 0,C 180,E1 -1082.711,E2 -1082.711} C_VEL
LIN {X 0,Y 594.394,Z 276.439,A -85,B 0,C 180,E1 -1085.428,E2 -1085.428} C_VEL
LIN {X 0,Y 594.411,Z 276.446,A -85,B 0,C 180,E1 -1088.157,E2 -1088.157} C_VEL
LIN {X 0,Y 594.386,Z 276.439,A -85,B 0,C 180,E1 -1091.071,E2 -1091.071} C_VEL
LIN {X 0,Y 594.38,Z 276.44,A -85,B 0,C 180,E1 -1093.679,E2 -1093.679} C_VEL
LIN {X 0,Y 594.392,Z 276.444,A -85,B 0,C 180,E1 -1096.718,E2 -1096.718} C_VEL
LIN {X 0,Y 594.367,Z 276.442,A -85,B 0,C 180,E1 -1099.334,E2 -1099.334} C_VEL
LIN {X 0,Y 594.363,Z 276.441,A -85,B 0,C 180,E1 -1101.503,E2 -1101.503} C_VEL
LIN {X 0,Y 594.39,Z 276.444,A -85,B 0,C 180,E1 -1104.446,E2 -1104.446} C_VEL
LIN {X 0,Y 594.381,Z 276.449,A -85,B 0,C 180,E1 -1106.7,E2 -1106.7} C_VEL
LIN {X 0,Y 594.382,Z 276.448,A -85,B 0,C 180,E1 -1108.998,E2 -1108.998} C_VEL
LIN {X 0,Y 594.377,Z 276.441,A -85,B 0,C 180,E1 -1111.642,E2 -1111.642} C_VEL
LIN {X 0,Y 594.376,Z 276.443,A -85,B 0,C 180,E1 -1114.58,E2 -1114.58} C_VEL
LIN {X 0,Y 594.391,Z 276.441,A -85,B 0,C 180,E1 -1117.608,E2 -1117.608} C_VEL
LIN {X 0,Y 594.368,Z 276.442,A -85,B 0,C 180,E1 -1120.567,E2 -1120.567} C_VEL
LIN {X 0,Y 594.368,Z 276.452,A -85,B 0,C 180,E1 -1123.299,E2 -1123.299} C_VEL
LIN {X 0,Y 594.361,Z 276.443,A -85,B 0,C 180,E1 -1126.161,E2 -1126.161} C_VEL
LIN {X 0,Y 594.381,Z 276.439,A -85,B 0,C 180,E1 -1128.536,E2 -1128.536} C_VEL
LIN {X 0,Y 594.381,Z 276.445,A -85,B 0,C 180,E1 -1131.296,E2 -1131.296} C_VEL
LIN {X 0,Y 594.352,Z 276.454,A -85,B 0,C 180,E1 -1133.755,E2 -1133.755} C_VEL
LIN {X 0,Y 594.366,Z 276.445,A -85,B 0,C 180,E1 -1136.238,E2 -1136.238} C_VEL
LIN {X 0,Y 594.37,Z 276.441,A -85,B 0,C 180,E1 -1138.65,E2 -1138.65} C_VEL
LIN {X 0,Y 594.384,Z 276.44,A -85,B 0,C 180,E1 -1141.042,E2 -1141.042} C_VEL
LIN {X 0,Y 594.381,Z 276.451,A -85,B 0,C 180,E1 -1143.979,E2 -1143.979} C_VEL
LIN {X 0,Y 594.386,Z 276.446,A -85,B 0,C 180,E1 -1146.665,E2 -1146.665} C_VEL
LIN {X 0,Y 594.403,Z 276.548,A -85,B 0,C 180,E1 -1146.988,E2 -1146.988} C_VEL
LIN {X 0,Y 594.766,Z 281.021,A -85,B 0,C 180,E1 -1147.637,E2 -1147.637} C_VEL
LIN {X 0,Y 594.637,Z 302.761,A -85,B 0,C 180,E1 -1150.674,E2 -1150.674} C_VEL
LIN {X 0,Y 594.554,Z 323.472,A -85,B 0,C 180,E1 -1153.519,E2 -1153.519} C_VEL
LIN {X 0,Y 594.439,Z 345.478,A -85,B 0,C 180,E1 -1156.496,E2 -1156.496} C_VEL
LIN {X 0,Y 594.442,Z 346.611,A -85,B 0,C 180,E1 -1156.649,E2 -1156.649} C_VEL
LIN {X 0,Y 594.776,Z 350.694,A -85,B 0,C 180,E1 -1156.722,E2 -1156.722} C_VEL
LIN {X 0,Y 594.646,Z 454.93,A -85,B 0,C 180,E1 -1157.998,E2 -1157.998} C_VEL
LIN {X 0,Y 594.621,Z 468.207,A -85,B 0,C 180,E1 -1158.3,E2 -1158.3} C_VEL
LIN {X 0,Y 594.574,Z 480.497,A -85,B 0,C 180,E1 -1158.715,E2 -1158.715} C_VEL
LIN {X 0,Y 594.533,Z 492.626,A -85,B 0,C 180,E1 -1159.27,E2 -1159.27} C_VEL
LIN {X 0,Y 594.46,Z 504.195,A -85,B 0,C 180,E1 -1159.957,E2 -1159.957} C_VEL
LIN {X 0,Y 594.413,Z 514.592,A -85,B 0,C 180,E1 -1160.729,E2 -1160.729} C_VEL
LIN {X 0,Y 594.349,Z 523.026,A -85,B 0,C 180,E1 -1161.5,E2 -1161.5} C_VEL
LIN {X 0,Y 594.347,Z 530.958,A -85,B 0,C 180,E1 -1162.355,E2 -1162.355} C_VEL
LIN {X 0,Y 594.281,Z 538.823,A -85,B 0,C 180,E1 -1163.41,E2 -1163.41} C_VEL
LIN {X 0,Y 594.289,Z 545.678,A -85,B 0,C 180,E1 -1164.571,E2 -1164.571} C_VEL
LIN {X 0,Y 594.27,Z 550.37,A -85,B 0,C 180,E1 -1165.591,E2 -1165.591} C_VEL
LIN {X 0,Y 594.267,Z 553.955,A -85,B 0,C 180,E1 -1166.61,E2 -1166.61} C_VEL
LIN {X 0,Y 594.226,Z 555.808,A -85,B 0,C 180,E1 -1167.288,E2 -1167.288} C_VEL
LIN {X 0,Y 594.24,Z 557.2,A -85,B 0,C 180,E1 -1167.966,E2 -1167.966} C_VEL
LIN {X 0,Y 594.239,Z 558.784,A -85,B 0,C 180,E1 -1169.322,E2 -1169.322} C_VEL
LIN {X 0,Y 594.236,Z 559,A -85,B 0,C 180,E1 -1170,E2 -1170} C_VEL
LIN {X 0,Y 594.247,Z 558.185,A -85,B 0,C 180,E1 -1171.355,E2 -1171.355} C_VEL
LIN {X 0,Y 594.24,Z 557.202,A -85,B 0,C 180,E1 -1172.033,E2 -1172.033} C_VEL
LIN {X 0,Y 594.226,Z 555.811,A -85,B 0,C 180,E1 -1172.711,E2 -1172.711} C_VEL
LIN {X 0,Y 594.288,Z 552.897,A -85,B 0,C 180,E1 -1173.729,E2 -1173.729} C_VEL
LIN {X 0,Y 594.241,Z 548.951,A -85,B 0,C 180,E1 -1174.748,E2 -1174.748} C_VEL
LIN {X 0,Y 594.304,Z 542.88,A -85,B 0,C 180,E1 -1175.939,E2 -1175.939} C_VEL
LIN {X 0,Y 594.307,Z 536.239,A -85,B 0,C 180,E1 -1176.962,E2 -1176.962} C_VEL
LIN {X 0,Y 594.359,Z 527.994,A -85,B 0,C 180,E1 -1177.986,E2 -1177.986} C_VEL
LIN {X 0,Y 594.404,Z 517.605,A -85,B 0,C 180,E1 -1179.013,E2 -1179.013} C_VEL
LIN {X 0,Y 594.448,Z 506.754,A -85,B 0,C 180,E1 -1179.87,E2 -1179.87} C_VEL
LIN {X 0,Y 594.505,Z 495.786,A -85,B 0,C 180,E1 -1180.558,E2 -1180.558} C_VEL
LIN {X 0,Y 594.566,Z 483.56,A -85,B 0,C 180,E1 -1181.158,E2 -1181.158} C_VEL
LIN {X 0,Y 594.579,Z 471.89,A -85,B 0,C 180,E1 -1181.592,E2 -1181.592} C_VEL
LIN {X 0,Y 594.633,Z 459.534,A -85,B 0,C 180,E1 -1181.915,E2 -1181.915} C_VEL
LIN {X 0,Y 594.689,Z 443.772,A -85,B 0,C 180,E1 -1182.152,E2 -1182.152} C_VEL
LIN {X 0,Y 594.625,Z 348.19,A -85,B 0,C 180,E1 -1183.312,E2 -1183.312} C_VEL
LIN {X 0,Y 594.423,Z 346.455,A -85,B 0,C 180,E1 -1183.373,E2 -1183.373} C_VEL
LIN {X 0,Y 594.478,Z 327.361,A -85,B 0,C 180,E1 -1185.953,E2 -1185.953} C_VEL
LIN {X 0,Y 594.584,Z 307.945,A -85,B 0,C 180,E1 -1188.61,E2 -1188.61} C_VEL
LIN {X 0,Y 594.707,Z 288.316,A -85,B 0,C 180,E1 -1191.338,E2 -1191.338} C_VEL
LIN {X 0,Y 594.672,Z 277.927,A -85,B 0,C 180,E1 -1192.805,E2 -1192.805} C_VEL
LIN {X 0,Y 594.391,Z 276.445,A -85,B 0,C 180,E1 -1193.058,E2 -1193.058} C_VEL
LIN {X 0,Y 594.371,Z 276.442,A -85,B 0,C 180,E1 -1195.193,E2 -1195.193} C_VEL
LIN {X 0,Y 594.386,Z 276.442,A -85,B 0,C 180,E1 -1197.526,E2 -1197.526} C_VEL
LIN {X 0,Y 594.385,Z 276.446,A -85,B 0,C 180,E1 -1200.328,E2 -1200.328} C_VEL
LIN {X 0,Y 594.375,Z 276.441,A -85,B 0,C 180,E1 -1202.95,E2 -1202.95} C_VEL
LIN {X 0,Y 594.347,Z 276.444,A -85,B 0,C 180,E1 -1205.408,E2 -1205.408} C_VEL
LIN {X 0,Y 594.383,Z 276.444,A -85,B 0,C 180,E1 -1207.94,E2 -1207.94} C_VEL
LIN {X 0,Y 594.376,Z 276.444,A -85,B 0,C 180,E1 -1210.822,E2 -1210.822} C_VEL
LIN {X 0,Y 594.364,Z 276.442,A -85,B 0,C 180,E1 -1213.299,E2 -1213.299} C_VEL
LIN {X 0,Y 594.364,Z 276.446,A -85,B 0,C 180,E1 -1216.16,E2 -1216.16} C_VEL
LIN {X 0,Y 594.38,Z 276.45,A -85,B 0,C 180,E1 -1218.536,E2 -1218.536} C_VEL
LIN {X 0,Y 594.383,Z 276.441,A -85,B 0,C 180,E1 -1221.295,E2 -1221.295} C_VEL
LIN {X 0,Y 594.39,Z 276.438,A -85,B 0,C 180,E1 -1223.758,E2 -1223.758} C_VEL
LIN {X 0,Y 594.375,Z 276.442,A -85,B 0,C 180,E1 -1226.238,E2 -1226.238} C_VEL
LIN {X 0,Y 594.386,Z 276.446,A -85,B 0,C 180,E1 -1228.651,E2 -1228.651} C_VEL
LIN {X 0,Y 594.377,Z 276.449,A -85,B 0,C 180,E1 -1231.042,E2 -1231.042} C_VEL
LIN {X 0,Y 594.384,Z 276.439,A -85,B 0,C 180,E1 -1233.976,E2 -1233.976} C_VEL
LIN {X 0,Y 594.384,Z 276.439,A -85,B 0,C 180,E1 -1236.296,E2 -1236.296} C_VEL
LIN {X 0,Y 594.398,Z 276.447,A -85,B 0,C 180,E1 -1239.224,E2 -1239.224} C_VEL
LIN {X 0,Y 594.346,Z 276.444,A -85,B 0,C 180,E1 -1242.095,E2 -1242.095} C_VEL
LIN {X 0,Y 594.359,Z 276.442,A -85,B 0,C 180,E1 -1244.219,E2 -1244.219} C_VEL
LIN {X 0,Y 594.365,Z 276.446,A -85,B 0,C 180,E1 -1247.017,E2 -1247.017} C_VEL
LIN {X 0,Y 594.383,Z 276.444,A -85,B 0,C 180,E1 -1249.784,E2 -1249.784} C_VEL
LIN {X 0,Y 594.395,Z 276.438,A -85,B 0,C 180,E1 -1252.527,E2 -1252.527} C_VEL
LIN {X 0,Y 594.392,Z 276.443,A -85,B 0,C 180,E1 -1255.253,E2 -1255.253} C_VEL
LIN {X 0,Y 594.381,Z 276.445,A -85,B 0,C 180,E1 -1257.967,E2 -1257.967} C_VEL
LIN {X 0,Y 594.405,Z 276.436,A -85,B 0,C 180,E1 -1260.678,E2 -1260.678} C_VEL
LIN {X 0,Y 594.385,Z 276.443,A -85,B 0,C 180,E1 -1263.389,E2 -1263.389} C_VEL
LIN {X 0,Y 594.362,Z 276.449,A -85,B 0,C 180,E1 -1266.109,E2 -1266.109} C_VEL
LIN {X 0,Y 594.407,Z 276.443,A -85,B 0,C 180,E1 -1268.157,E2 -1268.157} C_VEL
LIN {X 0,Y 594.374,Z 276.44,A -85,B 0,C 180,E1 -1271.069,E2 -1271.069} C_VEL
LIN {X 0,Y 594.375,Z 276.444,A -85,B 0,C 180,E1 -1273.679,E2 -1273.679} C_VEL
LIN {X 0,Y 594.343,Z 276.444,A -85,B 0,C 180,E1 -1275.308,E2 -1275.308} C_VEL
LIN {X 0,Y 593.678,Z 276.534,A -85,B 0,C 180,E1 -1275.874,E2 -1275.874} C_VEL
LIN {X 0,Y 590.818,Z 276.895,A -85,B 0,C 180,E1 -1276.792,E2 -1276.792} C_VEL
LIN {X 0,Y 588.405,Z 277.197,A -85,B 0,C 180,E1 -1277.531,E2 -1277.531} C_VEL
LIN {X 0,Y 587.378,Z 277.321,A -85,B 0,C 180,E1 -1278.101,E2 -1278.101} C_VEL
LIN {X 0,Y 587.3,Z 277.328,A -85,B 0,C 180,E1 -1278.294,E2 -1278.294} C_VEL
LIN {X 0,Y 587.326,Z 277.319,A -85,B 0,C 180,E1 -1281.038,E2 -1281.038} C_VEL
LIN {X 0,Y 587.309,Z 277.32,A -85,B 0,C 180,E1 -1283.26,E2 -1283.26} C_VEL
LIN {X 0,Y 587.323,Z 277.319,A -85,B 0,C 180,E1 -1285.518,E2 -1285.518} C_VEL
LIN {X 0,Y 587.317,Z 277.329,A -85,B 0,C 180,E1 -1288.598,E2 -1288.598} C_VEL
LIN {X 0,Y 587.32,Z 277.323,A -85,B 0,C 180,E1 -1290.968,E2 -1290.968} C_VEL
LIN {X 0,Y 587.323,Z 277.319,A -85,B 0,C 180,E1 -1293.398,E2 -1293.398} C_VEL
LIN {X 0,Y 587.286,Z 277.324,A -85,B 0,C 180,E1 -1295.901,E2 -1295.901} C_VEL
LIN {X 0,Y 587.323,Z 277.325,A -85,B 0,C 180,E1 -1298.48,E2 -1298.48} C_VEL
LIN {X 0,Y 587.327,Z 277.324,A -85,B 0,C 180,E1 -1301.158,E2 -1301.158} C_VEL
LIN {X 0,Y 587.3,Z 277.322,A -85,B 0,C 180,E1 -1304.112,E2 -1304.112} C_VEL
LIN {X 0,Y 587.296,Z 277.333,A -85,B 0,C 180,E1 -1306.993,E2 -1306.993} C_VEL
LIN {X 0,Y 587.302,Z 277.322,A -85,B 0,C 180,E1 -1309.746,E2 -1309.746} C_VEL
LIN {X 0,Y 587.337,Z 277.317,A -85,B 0,C 180,E1 -1312.393,E2 -1312.393} C_VEL
LIN {X 0,Y 587.336,Z 277.321,A -85,B 0,C 180,E1 -1315.655,E2 -1315.655} C_VEL
LIN {X 0,Y 587.332,Z 277.317,A -85,B 0,C 180,E1 -1318.231,E2 -1318.231} C_VEL
LIN {X 0,Y 587.341,Z 277.319,A -85,B 0,C 180,E1 -1320.869,E2 -1320.869} C_VEL
LIN {X 0,Y 587.296,Z 277.327,A -85,B 0,C 180,E1 -1323.833,E2 -1323.833} C_VEL
LIN {X 0,Y 587.303,Z 277.321,A -85,B 0,C 180,E1 -1326.741,E2 -1326.741} C_VEL
LIN {X 0,Y 587.32,Z 277.329,A -85,B 0,C 180,E1 -1329.695,E2 -1329.695} C_VEL
LIN {X 0,Y 587.287,Z 277.331,A -85,B 0,C 180,E1 -1331.873,E2 -1331.873} C_VEL
LIN {X 0,Y 587.298,Z 277.328,A -85,B 0,C 180,E1 -1334.025,E2 -1334.025} C_VEL
LIN {X 0,Y 587.336,Z 277.322,A -85,B 0,C 180,E1 -1336.154,E2 -1336.154} C_VEL
LIN {X 0,Y 587.294,Z 277.322,A -85,B 0,C 180,E1 -1338.962,E2 -1338.962} C_VEL
LIN {X 0,Y 587.323,Z 277.326,A -85,B 0,C 180,E1 -1341.745,E2 -1341.745} C_VEL
LIN {X 0,Y 587.323,Z 277.322,A -85,B 0,C 180,E1 -1344.507,E2 -1344.507} C_VEL
LIN {X 0,Y 587.333,Z 277.318,A -85,B 0,C 180,E1 -1347.257,E2 -1347.257} C_VEL
LIN {X 0,Y 587.382,Z 277.319,A -85,B 0,C 180,E1 -1350,E2 -1350} C_VEL
LIN {X 0,Y 587.339,Z 277.32,A -85,B 0,C 180,E1 -1352.744,E2 -1352.744} C_VEL
LIN {X 0,Y 587.312,Z 277.32,A -85,B 0,C 180,E1 -1355.494,E2 -1355.494} C_VEL
LIN {X 0,Y 587.314,Z 277.328,A -85,B 0,C 180,E1 -1358.256,E2 -1358.256} C_VEL
LIN {X 0,Y 587.287,Z 277.325,A -85,B 0,C 180,E1 -1361.1,E2 -1361.1} C_VEL
LIN {X 0,Y 587.311,Z 277.321,A -85,B 0,C 180,E1 -1363.847,E2 -1363.847} C_VEL
LIN {X 0,Y 587.312,Z 277.328,A -85,B 0,C 180,E1 -1366.8,E2 -1366.8} C_VEL
LIN {X 0,Y 587.29,Z 277.323,A -85,B 0,C 180,E1 -1369.577,E2 -1369.577} C_VEL
LIN {X 0,Y 587.267,Z 277.326,A -85,B 0,C 180,E1 -1371.777,E2 -1371.777} C_VEL
LIN {X 0,Y 587.283,Z 277.33,A -85,B 0,C 180,E1 -1374.564,E2 -1374.564} C_VEL
LIN {X 0,Y 587.293,Z 277.333,A -85,B 0,C 180,E1 -1377.048,E2 -1377.048} C_VEL
LIN {X 0,Y 587.297,Z 277.471,A -85,B 0,C 180,E1 -1378.112,E2 -1378.112} C_VEL
LIN {X 0,Y 587.389,Z 285.669,A -85,B 0,C 180,E1 -1379.574,E2 -1379.574} C_VEL
LIN {X 0,Y 587.346,Z 298.501,A -85,B 0,C 180,E1 -1381.835,E2 -1381.835} C_VEL
LIN {X 0,Y 587.327,Z 308.335,A -85,B 0,C 180,E1 -1383.551,E2 -1383.551} C_VEL
LIN {X 0,Y 587.861,Z 312.73,A -85,B 0,C 180,E1 -1383.633,E2 -1383.633} C_VEL
LIN {X 0,Y 587.746,Z 414.651,A -85,B 0,C 180,E1 -1384.896,E2 -1384.896} C_VEL
LIN {X 0,Y 587.672,Z 428.544,A -85,B 0,C 180,E1 -1385.214,E2 -1385.214} C_VEL
LIN {X 0,Y 587.563,Z 440.84,A -85,B 0,C 180,E1 -1385.639,E2 -1385.639} C_VEL
LIN {X 0,Y 587.521,Z 451.861,A -85,B 0,C 180,E1 -1386.149,E2 -1386.149} C_VEL
LIN {X 0,Y 587.456,Z 462.025,A -85,B 0,C 180,E1 -1386.739,E2 -1386.739} C_VEL
LIN {X 0,Y 587.404,Z 472.557,A -85,B 0,C 180,E1 -1387.495,E2 -1387.495} C_VEL
LIN {X 0,Y 587.336,Z 481.687,A -85,B 0,C 180,E1 -1388.305,E2 -1388.305} C_VEL
LIN {X 0,Y 587.294,Z 490.416,A -85,B 0,C 180,E1 -1389.243,E2 -1389.243} C_VEL
LIN {X 0,Y 587.221,Z 498.065,A -85,B 0,C 180,E1 -1390.262,E2 -1390.262} C_VEL
LIN {X 0,Y 587.202,Z 503.641,A -85,B 0,C 180,E1 -1391.169,E2 -1391.169} C_VEL
LIN {X 0,Y 587.195,Z 508.294,A -85,B 0,C 180,E1 -1392.092,E2 -1392.092} C_VEL
LIN {X 0,Y 587.165,Z 512.313,A -85,B 0,C 180,E1 -1393.102,E2 -1393.102} C_VEL
LIN {X 0,Y 587.164,Z 515.289,A -85,B 0,C 180,E1 -1394.096,E2 -1394.096} C_VEL
LIN {X 0,Y 587.156,Z 517.341,A -85,B 0,C 180,E1 -1395.073,E2 -1395.073} C_VEL
LIN {X 0,Y 587.14,Z 518.562,A -85,B 0,C 180,E1 -1396.032,E2 -1396.032} C_VEL
LIN {X 0,Y 587.166,Z 518.991,A -85,B 0,C 180,E1 -1396.979,E2 -1396.979} C_VEL
LIN {X 0,Y 587.167,Z 518.662,A -85,B 0,C 180,E1 -1397.911,E2 -1397.911} C_VEL
LIN {X 0,Y 587.125,Z 517.45,A -85,B 0,C 180,E1 -1398.949,E2 -1398.949} C_VEL
LIN {X 0,Y 587.151,Z 515.269,A -85,B 0,C 180,E1 -1400.001,E2 -1400.001} C_VEL
LIN {X 0,Y 587.169,Z 511.989,A -85,B 0,C 180,E1 -1401.078,E2 -1401.078} C_VEL
LIN {X 0,Y 587.177,Z 506.498,A -85,B 0,C 180,E1 -1402.379,E2 -1402.379} C_VEL
LIN {X 0,Y 587.224,Z 500.155,A -85,B 0,C 180,E1 -1403.505,E2 -1403.505} C_VEL
LIN {X 0,Y 587.237,Z 493.397,A -85,B 0,C 180,E1 -1404.471,E2 -1404.471} C_VEL
LIN {X 0,Y 587.298,Z 486.158,A -85,B 0,C 180,E1 -1405.326,E2 -1405.326} C_VEL
LIN {X 0,Y 587.336,Z 477.313,A -85,B 0,C 180,E1 -1406.191,E2 -1406.191} C_VEL
LIN {X 0,Y 587.41,Z 467.991,A -85,B 0,C 180,E1 -1406.942,E2 -1406.942} C_VEL
LIN {X 0,Y 587.475,Z 456.007,A -85,B 0,C 180,E1 -1407.718,E2 -1407.718} C_VEL
LIN {X 0,Y 587.555,Z 443.391,A -85,B 0,C 180,E1 -1408.344,E2 -1408.344} C_VEL
LIN {X 0,Y 587.634,Z 432.567,A -85,B 0,C 180,E1 -1408.751,E2 -1408.751} C_VEL
LIN {X 0,Y 587.642,Z 420.458,A -85,B 0,C 180,E1 -1409.08,E2 -1409.08} C_VEL
LIN {X 0,Y 587.692,Z 407.508,A -85,B 0,C 180,E1 -1409.298,E2 -1409.298} C_VEL
LIN {X 0,Y 587.821,Z 311.461,A -85,B 0,C 180,E1 -1410.474,E2 -1410.474} C_VEL
LIN {X 0,Y 587.342,Z 308.29,A -85,B 0,C 180,E1 -1410.546,E2 -1410.546} C_VEL
LIN {X 0,Y 587.386,Z 293.408,A -85,B 0,C 180,E1 -1413.149,E2 -1413.149} C_VEL
LIN {X 0,Y 587.468,Z 279.217,A -85,B 0,C 180,E1 -1415.661,E2 -1415.661} C_VEL
LIN {X 0,Y 587.37,Z 277.317,A -85,B 0,C 180,E1 -1416.042,E2 -1416.042} C_VEL
LIN {X 0,Y 587.333,Z 277.324,A -85,B 0,C 180,E1 -1418.962,E2 -1418.962} C_VEL
LIN {X 0,Y 587.306,Z 277.324,A -85,B 0,C 180,E1 -1421.872,E2 -1421.872} C_VEL
LIN {X 0,Y 587.321,Z 277.321,A -85,B 0,C 180,E1 -1424.024,E2 -1424.024} C_VEL
LIN {X 0,Y 587.358,Z 277.316,A -85,B 0,C 180,E1 -1426.154,E2 -1426.154} C_VEL
LIN {X 0,Y 587.342,Z 277.318,A -85,B 0,C 180,E1 -1428.962,E2 -1428.962} C_VEL
LIN {X 0,Y 587.342,Z 277.327,A -85,B 0,C 180,E1 -1431.744,E2 -1431.744} C_VEL
LIN {X 0,Y 587.356,Z 277.315,A -85,B 0,C 180,E1 -1434.507,E2 -1434.507} C_VEL
LIN {X 0,Y 587.37,Z 277.315,A -85,B 0,C 180,E1 -1437.257,E2 -1437.257} C_VEL
LIN {X 0,Y 587.383,Z 277.321,A -85,B 0,C 180,E1 -1440,E2 -1440} C_VEL
LIN {X 0,Y 587.366,Z 277.314,A -85,B 0,C 180,E1 -1442.743,E2 -1442.743} C_VEL
LIN {X 0,Y 587.358,Z 277.316,A -85,B 0,C 180,E1 -1445.493,E2 -1445.493} C_VEL
LIN {X 0,Y 587.363,Z 277.324,A -85,B 0,C 180,E1 -1448.255,E2 -1448.255} C_VEL
LIN {X 0,Y 587.35,Z 277.315,A -85,B 0,C 180,E1 -1451.134,E2 -1451.134} C_VEL
LIN {X 0,Y 587.366,Z 277.322,A -85,B 0,C 180,E1 -1454.26,E2 -1454.26} C_VEL
LIN {X 0,Y 587.345,Z 277.315,A -85,B 0,C 180,E1 -1457.406,E2 -1457.406} C_VEL
LIN {X 0,Y 587.314,Z 277.32,A -85,B 0,C 180,E1 -1459.576,E2 -1459.576} C_VEL
LIN {X 0,Y 587.339,Z 277.325,A -85,B 0,C 180,E1 -1462.514,E2 -1462.514} C_VEL
LIN {X 0,Y 587.332,Z 277.318,A -85,B 0,C 180,E1 -1465.517,E2 -1465.517} C_VEL
LIN {X 0,Y 587.341,Z 277.316,A -85,B 0,C 180,E1 -1467.818,E2 -1467.818} C_VEL
LIN {X 0,Y 587.338,Z 277.321,A -85,B 0,C 180,E1 -1470.51,E2 -1470.51} C_VEL
LIN {X 0,Y 587.328,Z 277.322,A -85,B 0,C 180,E1 -1473.397,E2 -1473.397} C_VEL
LIN {X 0,Y 587.291,Z 277.323,A -85,B 0,C 180,E1 -1475.9,E2 -1475.9} C_VEL
LIN {X 0,Y 587.33,Z 277.319,A -85,B 0,C 180,E1 -1478.479,E2 -1478.479} C_VEL
LIN {X 0,Y 587.336,Z 277.326,A -85,B 0,C 180,E1 -1481.157,E2 -1481.157} C_VEL
LIN {X 0,Y 587.314,Z 277.321,A -85,B 0,C 180,E1 -1484.112,E2 -1484.112} C_VEL
LIN {X 0,Y 587.315,Z 277.323,A -85,B 0,C 180,E1 -1486.993,E2 -1486.993} C_VEL
LIN {X 0,Y 587.312,Z 277.328,A -85,B 0,C 180,E1 -1489.745,E2 -1489.745} C_VEL
LIN {X 0,Y 587.345,Z 277.317,A -85,B 0,C 180,E1 -1492.392,E2 -1492.392} C_VEL
LIN {X 0,Y 587.343,Z 277.327,A -85,B 0,C 180,E1 -1495.653,E2 -1495.653} C_VEL
LIN {X 0,Y 587.342,Z 277.321,A -85,B 0,C 180,E1 -1498.231,E2 -1498.231} C_VEL
LIN {X 0,Y 587.351,Z 277.316,A -85,B 0,C 180,E1 -1500.867,E2 -1500.867} C_VEL
LIN {X 0,Y 587.341,Z 277.326,A -85,B 0,C 180,E1 -1503.823,E2 -1503.823} C_VEL
LIN {X 0,Y 587.339,Z 277.328,A -85,B 0,C 180,E1 -1505.993,E2 -1505.993} C_VEL
LIN {X 0,Y 587.356,Z 277.417,A -85,B 0,C 180,E1 -1506.821,E2 -1506.821} C_VEL
LIN {X 0,Y 587.86,Z 280.913,A -85,B 0,C 180,E1 -1507.344,E2 -1507.344} C_VEL
LIN {X 0,Y 587.698,Z 300.172,A -85,B 0,C 180,E1 -1510.073,E2 -1510.073} C_VEL
LIN {X 0,Y 587.569,Z 319.452,A -85,B 0,C 180,E1 -1512.761,E2 -1512.761} C_VEL
LIN {X 0,Y 587.451,Z 341.885,A -85,B 0,C 180,E1 -1515.843,E2 -1515.843} C_VEL
LIN {X 0,Y 587.392,Z 346.611,A -85,B 0,C 180,E1 -1516.485,E2 -1516.485} C_VEL
LIN {X 0,Y 587.87,Z 350.694,A -85,B 0,C 180,E1 -1516.563,E2 -1516.563} C_VEL
LIN {X 0,Y 587.725,Z 454.929,A -85,B 0,C 180,E1 -1517.855,E2 -1517.855} C_VEL
LIN {X 0,Y 587.672,Z 468.207,A -85,B 0,C 180,E1 -1518.16,E2 -1518.16} C_VEL
LIN {X 0,Y 587.603,Z 480.615,A -85,B 0,C 180,E1 -1518.584,E2 -1518.584} C_VEL
LIN {X 0,Y 587.549,Z 492.624,A -85,B 0,C 180,E1 -1519.141,E2 -1519.141} C_VEL
LIN {X 0,Y 587.443,Z 504.197,A -85,B 0,C 180,E1 -1519.836,E2 -1519.836} C_VEL
LIN {X 0,Y 587.392,Z 514.594,A -85,B 0,C 180,E1 -1520.617,E2 -1520.617} C_VEL
LIN {X 0,Y 587.299,Z 523.039,A -85,B 0,C 180,E1 -1521.397,E2 -1521.397} C_VEL
LIN {X 0,Y 587.274,Z 530.958,A -85,B 0,C 180,E1 -1522.262,E2 -1522.262} C_VEL
LIN {X 0,Y 587.23,Z 537.467,A -85,B 0,C 180,E1 -1523.126,E2 -1523.126} C_VEL
LIN {X 0,Y 587.236,Z 543.865,A -85,B 0,C 180,E1 -1524.161,E2 -1524.161} C_VEL
LIN {X 0,Y 587.147,Z 548.948,A -85,B 0,C 180,E1 -1525.193,E2 -1525.193} C_VEL
LIN {X 0,Y 587.212,Z 552.894,A -85,B 0,C 180,E1 -1526.225,E2 -1526.225} C_VEL
LIN {X 0,Y 587.132,Z 555.808,A -85,B 0,C 180,E1 -1527.255,E2 -1527.255} C_VEL
LIN {X 0,Y 587.139,Z 557.199,A -85,B 0,C 180,E1 -1527.942,E2 -1527.942} C_VEL
LIN {X 0,Y 587.14,Z 558.784,A -85,B 0,C 180,E1 -1529.314,E2 -1529.314} C_VEL
LIN {X 0,Y 587.137,Z 559,A -85,B 0,C 180,E1 -1530,E2 -1530} C_VEL
LIN {X 0,Y 587.147,Z 558.186,A -85,B 0,C 180,E1 -1531.371,E2 -1531.371} C_VEL
LIN {X 0,Y 587.139,Z 557.201,A -85,B 0,C 180,E1 -1532.058,E2 -1532.058} C_VEL
LIN {X 0,Y 587.132,Z 555.811,A -85,B 0,C 180,E1 -1532.744,E2 -1532.744} C_VEL
LIN {X 0,Y 587.212,Z 552.897,A -85,B 0,C 180,E1 -1533.774,E2 -1533.774} C_VEL
LIN {X 0,Y 587.147,Z 548.951,A -85,B 0,C 180,E1 -1534.806,E2 -1534.806} C_VEL
LIN {X 0,Y 587.217,Z 542.88,A -85,B 0,C 180,E1 -1536.011,E2 -1536.011} C_VEL
LIN {X 0,Y 587.244,Z 536.24,A -85,B 0,C 180,E1 -1537.046,E2 -1537.046} C_VEL
LIN {X 0,Y 587.297,Z 527.994,A -85,B 0,C 180,E1 -1538.083,E2 -1538.083} C_VEL
LIN {X 0,Y 587.357,Z 517.606,A -85,B 0,C 180,E1 -1539.122,E2 -1539.122} C_VEL
LIN {X 0,Y 587.444,Z 506.754,A -85,B 0,C 180,E1 -1539.989,E2 -1539.989} C_VEL
LIN {X 0,Y 587.521,Z 495.788,A -85,B 0,C 180,E1 -1540.685,E2 -1540.685} C_VEL
LIN {X 0,Y 587.601,Z 483.797,A -85,B 0,C 180,E1 -1541.282,E2 -1541.282} C_VEL
LIN {X 0,Y 587.637,Z 471.888,A -85,B 0,C 180,E1 -1541.73,E2 -1541.73} C_VEL
LIN {X 0,Y 587.688,Z 459.533,A -85,B 0,C 180,E1 -1542.058,E2 -1542.058} C_VEL
LIN {X 0,Y 587.744,Z 443.772,A -85,B 0,C 180,E1 -1542.297,E2 -1542.297} C_VEL
LIN {X 0,Y 587.719,Z 348.747,A -85,B 0,C 180,E1 -1543.465,E2 -1543.465} C_VEL
LIN {X 0,Y 587.392,Z 346.617,A -85,B 0,C 180,E1 -1543.514,E2 -1543.514} C_VEL
LIN {X 0,Y 587.47,Z 328.656,A -85,B 0,C 180,E1 -1545.971,E2 -1545.971} C_VEL
LIN {X 0,Y 587.608,Z 310.533,A -85,B 0,C 180,E1 -1548.478,E2 -1548.478} C_VEL
LIN {X 0,Y 587.787,Z 291.479,A -85,B 0,C 180,E1 -1551.152,E2 -1551.152} C_VEL
LIN {X 0,Y 587.806,Z 279.777,A -85,B 0,C 180,E1 -1552.821,E2 -1552.821} C_VEL
LIN {X 0,Y 587.334,Z 277.325,A -85,B 0,C 180,E1 -1553.205,E2 -1553.205} C_VEL
LIN {X 0,Y 587.33,Z 277.323,A -85,B 0,C 180,E1 -1555.516,E2 -1555.516} C_VEL
LIN {X 0,Y 587.348,Z 277.324,A -85,B 0,C 180,E1 -1557.817,E2 -1557.817} C_VEL
LIN {X 0,Y 587.336,Z 277.321,A -85,B 0,C 180,E1 -1560.509,E2 -1560.509} C_VEL
LIN {X 0,Y 587.331,Z 277.318,A -85,B 0,C 180,E1 -1563.396,E2 -1563.396} C_VEL
LIN {X 0,Y 587.289,Z 277.328,A -85,B 0,C 180,E1 -1565.899,E2 -1565.899} C_VEL
LIN {X 0,Y 587.326,Z 277.326,A -85,B 0,C 180,E1 -1568.479,E2 -1568.479} C_VEL
LIN {X 0,Y 587.334,Z 277.318,A -85,B 0,C 180,E1 -1571.156,E2 -1571.156} C_VEL
LIN {X 0,Y 587.323,Z 277.323,A -85,B 0,C 180,E1 -1574.113,E2 -1574.113} C_VEL
LIN {X 0,Y 587.312,Z 277.324,A -85,B 0,C 180,E1 -1576.993,E2 -1576.993} C_VEL
LIN {X 0,Y 587.314,Z 277.32,A -85,B 0,C 180,E1 -1579.746,E2 -1579.746} C_VEL
LIN {X 0,Y 587.342,Z 277.322,A -85,B 0,C 180,E1 -1582.392,E2 -1582.392} C_VEL
LIN {X 0,Y 587.321,Z 277.327,A -85,B 0,C 180,E1 -1584.944,E2 -1584.944} C_VEL
LIN {X 0,Y 587.334,Z 277.319,A -85,B 0,C 180,E1 -1587.421,E2 -1587.421} C_VEL
LIN {X 0,Y 587.33,Z 277.318,A -85,B 0,C 180,E1 -1589.83,E2 -1589.83} C_VEL
LIN {X 0,Y 587.346,Z 277.317,A -85,B 0,C 180,E1 -1592.307,E2 -1592.307} C_VEL
LIN {X 0,Y 587.332,Z 277.32,A -85,B 0,C 180,E1 -1594.483,E2 -1594.483} C_VEL
LIN {X 0,Y 587.314,Z 277.331,A -85,B 0,C 180,E1 -1597.131,E2 -1597.131} C_VEL
LIN {X 0,Y 587.323,Z 277.321,A -85,B 0,C 180,E1 -1599.695,E2 -1599.695} C_VEL
LIN {X 0,Y 587.344,Z 277.317,A -85,B 0,C 180,E1 -1602.594,E2 -1602.594} C_VEL
LIN {X 0,Y 587.358,Z 277.318,A -85,B 0,C 180,E1 -1605.74,E2 -1605.74} C_VEL
LIN {X 0,Y 587.342,Z 277.319,A -85,B 0,C 180,E1 -1608.866,E2 -1608.866} C_VEL
LIN {X 0,Y 587.362,Z 277.32,A -85,B 0,C 180,E1 -1611.745,E2 -1611.745} C_VEL
LIN {X 0,Y 587.352,Z 277.315,A -85,B 0,C 180,E1 -1614.507,E2 -1614.507} C_VEL
LIN {X 0,Y 587.373,Z 277.317,A -85,B 0,C 180,E1 -1617.257,E2 -1617.257} C_VEL
LIN {X 0,Y 587.372,Z 277.319,A -85,B 0,C 180,E1 -1620,E2 -1620} C_VEL
LIN {X 0,Y 587.36,Z 277.314,A -85,B 0,C 180,E1 -1622.743,E2 -1622.743} C_VEL
LIN {X 0,Y 587.36,Z 277.318,A -85,B 0,C 180,E1 -1625.493,E2 -1625.493} C_VEL
LIN {X 0,Y 587.358,Z 277.32,A -85,B 0,C 180,E1 -1628.256,E2 -1628.256} C_VEL
LIN {X 0,Y 587.342,Z 277.316,A -85,B 0,C 180,E1 -1631.134,E2 -1631.134} C_VEL
LIN {X 0,Y 587.353,Z 277.321,A -85,B 0,C 180,E1 -1633.846,E2 -1633.846} C_VEL
LIN {X 0,Y 587.334,Z 277.319,A -85,B 0,C 180,E1 -1636.812,E2 -1636.812} C_VEL
LIN {X 0,Y 587.3,Z 277.328,A -85,B 0,C 180,E1 -1638.294,E2 -1638.294} C_VEL
LIN {X 0,Y 586.655,Z 277.404,A -85,B 0,C 180,E1 -1638.866,E2 -1638.866} C_VEL
LIN {X 0,Y 583.834,Z 277.757,A -85,B 0,C 180,E1 -1639.795,E2 -1639.795} C_VEL
LIN {X 0,Y 581.427,Z 278.059,A -85,B 0,C 180,E1 -1640.542,E2 -1640.542} C_VEL
LIN {X 0,Y 580.374,Z 278.185,A -85,B 0,C 180,E1 -1641.118,E2 -1641.118} C_VEL
LIN {X 0,Y 580.279,Z 278.196,A -85,B 0,C 180,E1 -1641.313,E2 -1641.313} C_VEL
LIN {X 0,Y 580.293,Z 278.204,A -85,B 0,C 180,E1 -1644.317,E2 -1644.317} C_VEL
LIN {X 0,Y 580.261,Z 278.206,A -85,B 0,C 180,E1 -1646.625,E2 -1646.625} C_VEL
LIN {X 0,Y 580.293,Z 278.195,A -85,B 0,C 180,E1 -1649.31,E2 -1649.31} C_VEL
LIN {X 0,Y 580.294,Z 278.198,A -85,B 0,C 180,E1 -1652.201,E2 -1652.201} C_VEL
LIN {X 0,Y 580.283,Z 278.206,A -85,B 0,C 180,E1 -1654.697,E2 -1654.697} C_VEL
LIN {X 0,Y 580.292,Z 278.197,A -85,B 0,C 180,E1 -1657.269,E2 -1657.269} C_VEL
LIN {X 0,Y 580.283,Z 278.198,A -85,B 0,C 180,E1 -1660.271,E2 -1660.271} C_VEL
LIN {X 0,Y 580.271,Z 278.205,A -85,B 0,C 180,E1 -1662.707,E2 -1662.707} C_VEL
LIN {X 0,Y 580.253,Z 278.201,A -85,B 0,C 180,E1 -1665.611,E2 -1665.611} C_VEL
LIN {X 0,Y 580.272,Z 278.202,A -85,B 0,C 180,E1 -1668.671,E2 -1668.671} C_VEL
LIN {X 0,Y 580.266,Z 278.206,A -85,B 0,C 180,E1 -1670.965,E2 -1670.965} C_VEL
LIN {X 0,Y 580.247,Z 278.204,A -85,B 0,C 180,E1 -1673.596,E2 -1673.596} C_VEL
LIN {X 0,Y 580.275,Z 278.197,A -85,B 0,C 180,E1 -1676.143,E2 -1676.143} C_VEL
LIN {X 0,Y 580.264,Z 278.199,A -85,B 0,C 180,E1 -1678.615,E2 -1678.615} C_VEL
LIN {X 0,Y 580.282,Z 278.201,A -85,B 0,C 180,E1 -1681.024,E2 -1681.024} C_VEL
LIN {X 0,Y 580.254,Z 278.206,A -85,B 0,C 180,E1 -1683.675,E2 -1683.675} C_VEL
LIN {X 0,Y 580.256,Z 278.199,A -85,B 0,C 180,E1 -1686.442,E2 -1686.442} C_VEL
LIN {X 0,Y 580.27,Z 278.205,A -85,B 0,C 180,E1 -1689.438,E2 -1689.438} C_VEL
LIN {X 0,Y 580.251,Z 278.211,A -85,B 0,C 180,E1 -1691.645,E2 -1691.645} C_VEL
LIN {X 0,Y 580.276,Z 278.197,A -85,B 0,C 180,E1 -1694.547,E2 -1694.547} C_VEL
LIN {X 0,Y 580.246,Z 278.2,A -85,B 0,C 180,E1 -1696.696,E2 -1696.696} C_VEL
LIN {X 0,Y 580.272,Z 278.197,A -85,B 0,C 180,E1 -1698.827,E2 -1698.827} C_VEL
LIN {X 0,Y 580.294,Z 278.2,A -85,B 0,C 180,E1 -1701.644,E2 -1701.644} C_VEL
LIN {X 0,Y 580.293,Z 278.198,A -85,B 0,C 180,E1 -1704.44,E2 -1704.44} C_VEL
LIN {X 0,Y 580.302,Z 278.193,A -85,B 0,C 180,E1 -1707.224,E2 -1707.224} C_VEL
LIN {X 0,Y 580.351,Z 278.195,A -85,B 0,C 180,E1 -1710,E2 -1710} C_VEL
LIN {X 0,Y 580.306,Z 278.195,A -85,B 0,C 180,E1 -1712.777,E2 -1712.777} C_VEL
LIN {X 0,Y 580.282,Z 278.196,A -85,B 0,C 180,E1 -1715.561,E2 -1715.561} C_VEL
LIN {X 0,Y 580.287,Z 278.206,A -85,B 0,C 180,E1 -1718.357,E2 -1718.357} C_VEL
LIN {X 0,Y 580.238,Z 278.202,A -85,B 0,C 180,E1 -1721.175,E2 -1721.175} C_VEL
LIN {X 0,Y 580.276,Z 278.199,A -85,B 0,C 180,E1 -1724.018,E2 -1724.018} C_VEL
LIN {X 0,Y 580.273,Z 278.203,A -85,B 0,C 180,E1 -1726.899,E2 -1726.899} C_VEL
LIN {X 0,Y 580.253,Z 278.199,A -85,B 0,C 180,E1 -1729.824,E2 -1729.824} C_VEL
LIN {X 0,Y 580.222,Z 278.205,A -85,B 0,C 180,E1 -1732.055,E2 -1732.055} C_VEL
LIN {X 0,Y 580.237,Z 278.211,A -85,B 0,C 180,E1 -1734.711,E2 -1734.711} C_VEL
LIN {X 0,Y 580.23,Z 278.209,A -85,B 0,C 180,E1 -1737.405,E2 -1737.405} C_VEL
LIN {X 0,Y 580.281,Z 278.347,A -85,B 0,C 180,E1 -1738.033,E2 -1738.033} C_VEL
LIN {X 0,Y 580.448,Z 285.534,A -85,B 0,C 180,E1 -1739.334,E2 -1739.334} C_VEL
LIN {X 0,Y 580.32,Z 298.84,A -85,B 0,C 180,E1 -1741.706,E2 -1741.706} C_VEL
LIN {X 0,Y 580.308,Z 308.531,A -85,B 0,C 180,E1 -1743.402,E2 -1743.402} C_VEL
LIN {X 0,Y 580.962,Z 312.917,A -85,B 0,C 180,E1 -1743.473,E2 -1743.473} C_VEL
LIN {X 0,Y 580.804,Z 415.714,A -85,B 0,C 180,E1 -1744.767,E2 -1744.767} C_VEL
LIN {X 0,Y 580.705,Z 429.227,A -85,B 0,C 180,E1 -1745.091,E2 -1745.091} C_VEL
LIN {X 0,Y 580.609,Z 441.319,A -85,B 0,C 180,E1 -1745.522,E2 -1745.522} C_VEL
LIN {X 0,Y 580.532,Z 452.671,A -85,B 0,C 180,E1 -1746.06,E2 -1746.06} C_VEL
LIN {X 0,Y 580.439,Z 463.121,A -85,B 0,C 180,E1 -1746.685,E2 -1746.685} C_VEL
LIN {X 0,Y 580.345,Z 473.833,A -85,B 0,C 180,E1 -1747.483,E2 -1747.483} C_VEL
LIN {X 0,Y 580.268,Z 483.361,A -85,B 0,C 180,E1 -1748.369,E2 -1748.369} C_VEL
LIN {X 0,Y 580.201,Z 491.832,A -85,B 0,C 180,E1 -1749.327,E2 -1749.327} C_VEL
LIN {X 0,Y 580.141,Z 498.527,A -85,B 0,C 180,E1 -1750.252,E2 -1750.252} C_VEL
LIN {X 0,Y 580.13,Z 504.764,A -85,B 0,C 180,E1 -1751.314,E2 -1751.314} C_VEL
LIN {X 0,Y 580.094,Z 509.62,A -85,B 0,C 180,E1 -1752.35,E2 -1752.35} C_VEL
LIN {X 0,Y 580.059,Z 513.311,A -85,B 0,C 180,E1 -1753.367,E2 -1753.367} C_VEL
LIN {X 0,Y 580.066,Z 516.599,A -85,B 0,C 180,E1 -1754.646,E2 -1754.646} C_VEL
LIN {X 0,Y 580.045,Z 518.155,A -85,B 0,C 180,E1 -1755.632,E2 -1755.632} C_VEL
LIN {X 0,Y 580.033,Z 518.898,A -85,B 0,C 180,E1 -1756.635,E2 -1756.635} C_VEL
LIN {X 0,Y 580.068,Z 518.811,A -85,B 0,C 180,E1 -1757.652,E2 -1757.652} C_VEL
LIN {X 0,Y 580.039,Z 517.84,A -85,B 0,C 180,E1 -1758.696,E2 -1758.696} C_VEL
LIN {X 0,Y 580.058,Z 515.246,A -85,B 0,C 180,E1 -1760.047,E2 -1760.047} C_VEL
LIN {X 0,Y 580.057,Z 511.04,A -85,B 0,C 180,E1 -1761.392,E2 -1761.392} C_VEL
LIN {X 0,Y 580.096,Z 507.025,A -85,B 0,C 180,E1 -1762.334,E2 -1762.334} C_VEL
LIN {X 0,Y 580.159,Z 501.665,A -85,B 0,C 180,E1 -1763.341,E2 -1763.341} C_VEL
LIN {X 0,Y 580.164,Z 494.273,A -85,B 0,C 180,E1 -1764.446,E2 -1764.446} C_VEL
LIN {X 0,Y 580.241,Z 485.937,A -85,B 0,C 180,E1 -1765.45,E2 -1765.45} C_VEL
LIN {X 0,Y 580.318,Z 477.425,A -85,B 0,C 180,E1 -1766.292,E2 -1766.292} C_VEL
LIN {X 0,Y 580.38,Z 467.718,A -85,B 0,C 180,E1 -1767.084,E2 -1767.084} C_VEL
LIN {X 0,Y 580.486,Z 455.561,A -85,B 0,C 180,E1 -1767.874,E2 -1767.874} C_VEL
LIN {X 0,Y 580.592,Z 443.386,A -85,B 0,C 180,E1 -1768.481,E2 -1768.481} C_VEL
LIN {X 0,Y 580.668,Z 432.614,A -85,B 0,C 180,E1 -1768.89,E2 -1768.89} C_VEL
LIN {X 0,Y 580.706,Z 421.934,A -85,B 0,C 180,E1 -1769.191,E2 -1769.191} C_VEL
LIN {X 0,Y 580.771,Z 410.238,A -85,B 0,C 180,E1 -1769.41,E2 -1769.41} C_VEL
LIN {X 0,Y 580.856,Z 311.756,A -85,B 0,C 180,E1 -1770.634,E2 -1770.634} C_VEL
LIN {X 0,Y 580.29,Z 308.408,A -85,B 0,C 180,E1 -1770.693,E2 -1770.693} C_VEL
LIN {X 0,Y 580.386,Z 293.22,A -85,B 0,C 180,E1 -1773.382,E2 -1773.382} C_VEL
LIN {X 0,Y 580.424,Z 279.305,A -85,B 0,C 180,E1 -1775.879,E2 -1775.879} C_VEL
LIN {X 0,Y 580.317,Z 278.196,A -85,B 0,C 180,E1 -1776.112,E2 -1776.112} C_VEL
LIN {X 0,Y 580.303,Z 278.198,A -85,B 0,C 180,E1 -1778.834,E2 -1778.834} C_VEL
LIN {X 0,Y 580.266,Z 278.205,A -85,B 0,C 180,E1 -1781.645,E2 -1781.645} C_VEL
LIN {X 0,Y 580.277,Z 278.201,A -85,B 0,C 180,E1 -1783.825,E2 -1783.825} C_VEL
LIN {X 0,Y 580.326,Z 278.194,A -85,B 0,C 180,E1 -1785.983,E2 -1785.983} C_VEL
LIN {X 0,Y 580.307,Z 278.194,A -85,B 0,C 180,E1 -1788.827,E2 -1788.827} C_VEL
LIN {X 0,Y 580.312,Z 278.203,A -85,B 0,C 180,E1 -1791.643,E2 -1791.643} C_VEL
LIN {X 0,Y 580.276,Z 278.208,A -85,B 0,C 180,E1 -1793.742,E2 -1793.742} C_VEL
LIN {X 0,Y 580.266,Z 278.209,A -85,B 0,C 180,E1 -1795.832,E2 -1795.832} C_VEL
LIN {X 0,Y 580.336,Z 278.199,A -85,B 0,C 180,E1 -1797.918,E2 -1797.918} C_VEL
LIN {X 0,Y 580.357,Z 278.187,A -85,B 0,C 180,E1 -1800.694,E2 -1800.694} C_VEL
LIN {X 0,Y 580.286,Z 278.197,A -85,B 0,C 180,E1 -1803.472,E2 -1803.472} C_VEL
LIN {X 0,Y 580.323,Z 278.193,A -85,B 0,C 180,E1 -1805.56,E2 -1805.56} C_VEL
LIN {X 0,Y 580.327,Z 278.199,A -85,B 0,C 180,E1 -1808.356,E2 -1808.356} C_VEL
LIN {X 0,Y 580.302,Z 278.193,A -85,B 0,C 180,E1 -1811.191,E2 -1811.191} C_VEL
LIN {X 0,Y 580.326,Z 278.194,A -85,B 0,C 180,E1 -1814.017,E2 -1814.017} C_VEL
LIN {X 0,Y 580.314,Z 278.195,A -85,B 0,C 180,E1 -1816.914,E2 -1816.914} C_VEL
LIN {X 0,Y 580.288,Z 278.196,A -85,B 0,C 180,E1 -1819.823,E2 -1819.823} C_VEL
LIN {X 0,Y 580.271,Z 278.199,A -85,B 0,C 180,E1 -1822.053,E2 -1822.053} C_VEL
LIN {X 0,Y 580.306,Z 278.198,A -85,B 0,C 180,E1 -1825.08,E2 -1825.08} C_VEL
LIN {X 0,Y 580.297,Z 278.194,A -85,B 0,C 180,E1 -1828.186,E2 -1828.186} C_VEL
LIN {X 0,Y 580.285,Z 278.202,A -85,B 0,C 180,E1 -1830.694,E2 -1830.694} C_VEL
LIN {X 0,Y 580.284,Z 278.201,A -85,B 0,C 180,E1 -1833.313,E2 -1833.313} C_VEL
LIN {X 0,Y 580.246,Z 278.202,A -85,B 0,C 180,E1 -1835.756,E2 -1835.756} C_VEL
LIN {X 0,Y 580.289,Z 278.195,A -85,B 0,C 180,E1 -1838.146,E2 -1838.146} C_VEL
LIN {X 0,Y 580.299,Z 278.198,A -85,B 0,C 180,E1 -1840.844,E2 -1840.844} C_VEL
LIN {X 0,Y 580.275,Z 278.202,A -85,B 0,C 180,E1 -1843.658,E2 -1843.658} C_VEL
LIN {X 0,Y 580.276,Z 278.197,A -85,B 0,C 180,E1 -1846.61,E2 -1846.61} C_VEL
LIN {X 0,Y 580.299,Z 278.198,A -85,B 0,C 180,E1 -1849.156,E2 -1849.156} C_VEL
LIN {X 0,Y 580.29,Z 278.201,A -85,B 0,C 180,E1 -1851.927,E2 -1851.927} C_VEL
LIN {X 0,Y 580.252,Z 278.201,A -85,B 0,C 180,E1 -1854.452,E2 -1854.452} C_VEL
LIN {X 0,Y 580.291,Z 278.196,A -85,B 0,C 180,E1 -1856.975,E2 -1856.975} C_VEL
LIN {X 0,Y 580.298,Z 278.198,A -85,B 0,C 180,E1 -1859.425,E2 -1859.425} C_VEL
LIN {X 0,Y 580.294,Z 278.203,A -85,B 0,C 180,E1 -1862.142,E2 -1862.142} C_VEL
LIN {X 0,Y 580.323,Z 278.193,A -85,B 0,C 180,E1 -1865.27,E2 -1865.27} C_VEL
LIN {X 0,Y 580.311,Z 278.22,A -85,B 0,C 180,E1 -1866.659,E2 -1866.659} C_VEL
LIN {X 0,Y 580.936,Z 283.344,A -85,B 0,C 180,E1 -1867.412,E2 -1867.412} C_VEL
LIN {X 0,Y 580.752,Z 302.761,A -85,B 0,C 180,E1 -1870.193,E2 -1870.193} C_VEL
LIN {X 0,Y 580.57,Z 322.714,A -85,B 0,C 180,E1 -1873.004,E2 -1873.004} C_VEL
LIN {X 0,Y 580.423,Z 345.478,A -85,B 0,C 180,E1 -1876.164,E2 -1876.164} C_VEL
LIN {X 0,Y 580.398,Z 346.611,A -85,B 0,C 180,E1 -1876.319,E2 -1876.319} C_VEL
LIN {X 0,Y 580.962,Z 352.482,A -85,B 0,C 180,E1 -1876.422,E2 -1876.422} C_VEL
LIN {X 0,Y 580.787,Z 454.929,A -85,B 0,C 180,E1 -1877.707,E2 -1877.707} C_VEL
LIN {X 0,Y 580.73,Z 468.208,A -85,B 0,C 180,E1 -1878.016,E2 -1878.016} C_VEL
LIN {X 0,Y 580.629,Z 480.365,A -85,B 0,C 180,E1 -1878.435,E2 -1878.435} C_VEL
LIN {X 0,Y 580.556,Z 492.623,A -85,B 0,C 180,E1 -1879.008,E2 -1879.008} C_VEL
LIN {X 0,Y 580.421,Z 504.198,A -85,B 0,C 180,E1 -1879.711,E2 -1879.711} C_VEL
LIN {X 0,Y 580.343,Z 514.595,A -85,B 0,C 180,E1 -1880.502,E2 -1880.502} C_VEL
LIN {X 0,Y 580.263,Z 523.053,A -85,B 0,C 180,E1 -1881.292,E2 -1881.292} C_VEL
LIN {X 0,Y 580.222,Z 530.958,A -85,B 0,C 180,E1 -1882.168,E2 -1882.168} C_VEL
LIN {X 0,Y 580.156,Z 538.634,A -85,B 0,C 180,E1 -1883.219,E2 -1883.219} C_VEL
LIN {X 0,Y 580.139,Z 545.678,A -85,B 0,C 180,E1 -1884.438,E2 -1884.438} C_VEL
LIN {X 0,Y 580.108,Z 550.37,A -85,B 0,C 180,E1 -1885.483,E2 -1885.483} C_VEL
LIN {X 0,Y 580.123,Z 553.956,A -85,B 0,C 180,E1 -1886.527,E2 -1886.527} C_VEL
LIN {X 0,Y 580.043,Z 555.807,A -85,B 0,C 180,E1 -1887.222,E2 -1887.222} C_VEL
LIN {X 0,Y 580.038,Z 557.198,A -85,B 0,C 180,E1 -1887.916,E2 -1887.916} C_VEL
LIN {X 0,Y 580.04,Z 558.784,A -85,B 0,C 180,E1 -1889.305,E2 -1889.305} C_VEL
LIN {X 0,Y 580.037,Z 559,A -85,B 0,C 180,E1 -1890,E2 -1890} C_VEL
LIN {X 0,Y 580.046,Z 558.186,A -85,B 0,C 180,E1 -1891.388,E2 -1891.388} C_VEL
LIN {X 0,Y 580.038,Z 557.201,A -85,B 0,C 180,E1 -1892.083,E2 -1892.083} C_VEL
LIN {X 0,Y 580.043,Z 555.811,A -85,B 0,C 180,E1 -1892.778,E2 -1892.778} C_VEL
LIN {X 0,Y 580.109,Z 552.897,A -85,B 0,C 180,E1 -1893.82,E2 -1893.82} C_VEL
LIN {X 0,Y 580.053,Z 548.951,A -85,B 0,C 180,E1 -1894.865,E2 -1894.865} C_VEL
LIN {X 0,Y 580.14,Z 542.88,A -85,B 0,C 180,E1 -1896.084,E2 -1896.084} C_VEL
LIN {X 0,Y 580.183,Z 536.241,A -85,B 0,C 180,E1 -1897.132,E2 -1897.132} C_VEL
LIN {X 0,Y 580.246,Z 527.994,A -85,B 0,C 180,E1 -1898.181,E2 -1898.181} C_VEL
LIN {X 0,Y 580.332,Z 517.607,A -85,B 0,C 180,E1 -1899.233,E2 -1899.233} C_VEL
LIN {X 0,Y 580.43,Z 507.933,A -85,B 0,C 180,E1 -1900.023,E2 -1900.023} C_VEL
LIN {X 0,Y 580.531,Z 497.335,A -85,B 0,C 180,E1 -1900.727,E2 -1900.727} C_VEL
LIN {X 0,Y 580.612,Z 485.486,A -85,B 0,C 180,E1 -1901.344,E2 -1901.344} C_VEL
LIN {X 0,Y 580.67,Z 473.188,A -85,B 0,C 180,E1 -1901.829,E2 -1901.829} C_VEL
LIN {X 0,Y 580.754,Z 460.54,A -85,B 0,C 180,E1 -1902.182,E2 -1902.182} C_VEL
LIN {X 0,Y 580.834,Z 447.35,A -85,B 0,C 180,E1 -1902.402,E2 -1902.402} C_VEL
LIN {X 0,Y 580.805,Z 349.42,A -85,B 0,C 180,E1 -1903.62,E2 -1903.62} C_VEL
LIN {X 0,Y 580.398,Z 346.617,A -85,B 0,C 180,E1 -1903.68,E2 -1903.68} C_VEL
LIN {X 0,Y 580.544,Z 326.067,A -85,B 0,C 180,E1 -1906.528,E2 -1906.528} C_VEL
LIN {X 0,Y 580.754,Z 305.061,A -85,B 0,C 180,E1 -1909.48,E2 -1909.48} C_VEL
LIN {X 0,Y 580.973,Z 283.35,A -85,B 0,C 180,E1 -1912.586,E2 -1912.586} C_VEL
LIN {X 0,Y 580.311,Z 278.201,A -85,B 0,C 180,E1 -1913.377,E2 -1913.377} C_VEL
LIN {X 0,Y 580.281,Z 278.207,A -85,B 0,C 180,E1 -1915.849,E2 -1915.849} C_VEL
LIN {X 0,Y 580.3,Z 278.202,A -85,B 0,C 180,E1 -1918.185,E2 -1918.185} C_VEL
LIN {X 0,Y 580.284,Z 278.197,A -85,B 0,C 180,E1 -1920.694,E2 -1920.694} C_VEL
LIN {X 0,Y 580.301,Z 278.194,A -85,B 0,C 180,E1 -1923.316,E2 -1923.316} C_VEL
LIN {X 0,Y 580.243,Z 278.204,A -85,B 0,C 180,E1 -1925.756,E2 -1925.756} C_VEL
LIN {X 0,Y 580.286,Z 278.203,A -85,B 0,C 180,E1 -1928.146,E2 -1928.146} C_VEL
LIN {X 0,Y 580.296,Z 278.197,A -85,B 0,C 180,E1 -1930.843,E2 -1930.843} C_VEL
LIN {X 0,Y 580.276,Z 278.197,A -85,B 0,C 180,E1 -1933.657,E2 -1933.657} C_VEL
LIN {X 0,Y 580.274,Z 278.207,A -85,B 0,C 180,E1 -1936.609,E2 -1936.609} C_VEL
LIN {X 0,Y 580.296,Z 278.196,A -85,B 0,C 180,E1 -1939.156,E2 -1939.156} C_VEL
LIN {X 0,Y 580.287,Z 278.196,A -85,B 0,C 180,E1 -1941.926,E2 -1941.926} C_VEL
LIN {X 0,Y 580.281,Z 278.202,A -85,B 0,C 180,E1 -1944.455,E2 -1944.455} C_VEL
LIN {X 0,Y 580.286,Z 278.204,A -85,B 0,C 180,E1 -1946.975,E2 -1946.975} C_VEL
LIN {X 0,Y 580.298,Z 278.196,A -85,B 0,C 180,E1 -1949.425,E2 -1949.425} C_VEL
LIN {X 0,Y 580.293,Z 278.195,A -85,B 0,C 180,E1 -1952.141,E2 -1952.141} C_VEL
LIN {X 0,Y 580.316,Z 278.198,A -85,B 0,C 180,E1 -1955.269,E2 -1955.269} C_VEL
LIN {X 0,Y 580.265,Z 278.198,A -85,B 0,C 180,E1 -1957.947,E2 -1957.947} C_VEL
LIN {X 0,Y 580.313,Z 278.198,A -85,B 0,C 180,E1 -1960.914,E2 -1960.914} C_VEL
LIN {X 0,Y 580.271,Z 278.199,A -85,B 0,C 180,E1 -1963.825,E2 -1963.825} C_VEL
LIN {X 0,Y 580.319,Z 278.193,A -85,B 0,C 180,E1 -1965.983,E2 -1965.983} C_VEL
LIN {X 0,Y 580.298,Z 278.196,A -85,B 0,C 180,E1 -1968.827,E2 -1968.827} C_VEL
LIN {X 0,Y 580.327,Z 278.199,A -85,B 0,C 180,E1 -1971.644,E2 -1971.644} C_VEL
LIN {X 0,Y 580.317,Z 278.192,A -85,B 0,C 180,E1 -1974.44,E2 -1974.44} C_VEL
LIN {X 0,Y 580.339,Z 278.193,A -85,B 0,C 180,E1 -1977.224,E2 -1977.224} C_VEL
LIN {X 0,Y 580.341,Z 278.194,A -85,B 0,C 180,E1 -1980,E2 -1980} C_VEL
LIN {X 0,Y 580.327,Z 278.19,A -85,B 0,C 180,E1 -1982.777,E2 -1982.777} C_VEL
LIN {X 0,Y 580.324,Z 278.196,A -85,B 0,C 180,E1 -1985.56,E2 -1985.56} C_VEL
LIN {X 0,Y 580.321,Z 278.195,A -85,B 0,C 180,E1 -1988.356,E2 -1988.356} C_VEL
LIN {X 0,Y 580.294,Z 278.194,A -85,B 0,C 180,E1 -1991.191,E2 -1991.191} C_VEL
LIN {X 0,Y 580.31,Z 278.202,A -85,B 0,C 180,E1 -1994.018,E2 -1994.018} C_VEL
LIN {X 0,Y 580.307,Z 278.193,A -85,B 0,C 180,E1 -1996.914,E2 -1996.914} C_VEL
LIN {X 0,Y 580.281,Z 278.199,A -85,B 0,C 180,E1 -1999.823,E2 -1999.823} C_VEL
LIN {X 0,Y 580.279,Z 278.196,A -85,B 0,C 180,E1 -2001.313,E2 -2001.313} C_VEL
LIN {X 0,Y 579.579,Z 278.289,A -85,B 0,C 180,E1 -2001.892,E2 -2001.892} C_VEL
LIN {X 0,Y 576.701,Z 278.645,A -85,B 0,C 180,E1 -2002.832,E2 -2002.832} C_VEL
LIN {X 0,Y 574.306,Z 278.942,A -85,B 0,C 180,E1 -2003.588,E2 -2003.588} C_VEL
LIN {X 0,Y 573.308,Z 279.072,A -85,B 0,C 180,E1 -2004.172,E2 -2004.172} C_VEL
LIN {X 0,Y 573.241,Z 279.077,A -85,B 0,C 180,E1 -2004.37,E2 -2004.37} C_VEL
LIN {X 0,Y 573.198,Z 279.081,A -85,B 0,C 180,E1 -2006.979,E2 -2006.979} C_VEL
LIN {X 0,Y 573.239,Z 279.073,A -85,B 0,C 180,E1 -2009.488,E2 -2009.488} C_VEL
LIN {X 0,Y 573.249,Z 279.083,A -85,B 0,C 180,E1 -2012.646,E2 -2012.646} C_VEL
LIN {X 0,Y 573.201,Z 279.081,A -85,B 0,C 180,E1 -2015.189,E2 -2015.189} C_VEL
LIN {X 0,Y 573.23,Z 279.074,A -85,B 0,C 180,E1 -2017.808,E2 -2017.808} C_VEL
LIN {X 0,Y 573.242,Z 279.078,A -85,B 0,C 180,E1 -2020.526,E2 -2020.526} C_VEL
LIN {X 0,Y 573.207,Z 279.08,A -85,B 0,C 180,E1 -2023.363,E2 -2023.363} C_VEL
LIN {X 0,Y 573.234,Z 279.075,A -85,B 0,C 180,E1 -2026.333,E2 -2026.333} C_VEL
LIN {X 0,Y 573.244,Z 279.076,A -85,B 0,C 180,E1 -2029.476,E2 -2029.476} C_VEL
LIN {X 0,Y 573.226,Z 279.075,A -85,B 0,C 180,E1 -2032.193,E2 -2032.193} C_VEL
LIN {X 0,Y 573.232,Z 279.085,A -85,B 0,C 180,E1 -2035.23,E2 -2035.23} C_VEL
LIN {X 0,Y 573.225,Z 279.075,A -85,B 0,C 180,E1 -2038.184,E2 -2038.184} C_VEL
LIN {X 0,Y 573.233,Z 279.075,A -85,B 0,C 180,E1 -2040.633,E2 -2040.633} C_VEL
LIN {X 0,Y 573.2,Z 279.088,A -85,B 0,C 180,E1 -2043.516,E2 -2043.516} C_VEL
LIN {X 0,Y 573.206,Z 279.079,A -85,B 0,C 180,E1 -2046.134,E2 -2046.134} C_VEL
LIN {X 0,Y 573.254,Z 279.071,A -85,B 0,C 180,E1 -2048.71,E2 -2048.71} C_VEL
LIN {X 0,Y 573.203,Z 279.084,A -85,B 0,C 180,E1 -2051.411,E2 -2051.411} C_VEL
LIN {X 0,Y 573.223,Z 279.084,A -85,B 0,C 180,E1 -2053.621,E2 -2053.621} C_VEL
LIN {X 0,Y 573.264,Z 279.081,A -85,B 0,C 180,E1 -2055.807,E2 -2055.807} C_VEL
LIN {X 0,Y 573.231,Z 279.074,A -85,B 0,C 180,E1 -2058.765,E2 -2058.765} C_VEL
LIN {X 0,Y 573.238,Z 279.077,A -85,B 0,C 180,E1 -2061.54,E2 -2061.54} C_VEL
LIN {X 0,Y 573.263,Z 279.075,A -85,B 0,C 180,E1 -2064.372,E2 -2064.372} C_VEL
LIN {X 0,Y 573.309,Z 279.071,A -85,B 0,C 180,E1 -2067.893,E2 -2067.893} C_VEL
LIN {X 0,Y 573.32,Z 279.071,A -85,B 0,C 180,E1 -2070,E2 -2070} C_VEL
LIN {X 0,Y 573.273,Z 279.071,A -85,B 0,C 180,E1 -2072.811,E2 -2072.811} C_VEL
LIN {X 0,Y 573.253,Z 279.072,A -85,B 0,C 180,E1 -2075.629,E2 -2075.629} C_VEL
LIN {X 0,Y 573.231,Z 279.084,A -85,B 0,C 180,E1 -2078.461,E2 -2078.461} C_VEL
LIN {X 0,Y 573.202,Z 279.078,A -85,B 0,C 180,E1 -2081.314,E2 -2081.314} C_VEL
LIN {X 0,Y 573.226,Z 279.079,A -85,B 0,C 180,E1 -2084.194,E2 -2084.194} C_VEL
LIN {X 0,Y 573.221,Z 279.078,A -85,B 0,C 180,E1 -2087.113,E2 -2087.113} C_VEL
LIN {X 0,Y 573.198,Z 279.08,A -85,B 0,C 180,E1 -2090.079,E2 -2090.079} C_VEL
LIN {X 0,Y 573.203,Z 279.082,A -85,B 0,C 180,E1 -2092.339,E2 -2092.339} C_VEL
LIN {X 0,Y 573.187,Z 279.084,A -85,B 0,C 180,E1 -2095.414,E2 -2095.414} C_VEL
LIN {X 0,Y 573.22,Z 279.223,A -85,B 0,C 180,E1 -2097.95,E2 -2097.95} C_VEL
LIN {X 0,Y 573.448,Z 285.774,A -85,B 0,C 180,E1 -2099.155,E2 -2099.155} C_VEL
LIN {X 0,Y 573.312,Z 299.344,A -85,B 0,C 180,E1 -2101.605,E2 -2101.605} C_VEL
LIN {X 0,Y 573.262,Z 308.37,A -85,B 0,C 180,E1 -2103.22,E2 -2103.22} C_VEL
LIN {X 0,Y 574.059,Z 314.433,A -85,B 0,C 180,E1 -2103.325,E2 -2103.325} C_VEL
LIN {X 0,Y 573.891,Z 415.42,A -85,B 0,C 180,E1 -2104.611,E2 -2104.611} C_VEL
LIN {X 0,Y 573.781,Z 427.946,A -85,B 0,C 180,E1 -2104.906,E2 -2104.906} C_VEL
LIN {X 0,Y 573.697,Z 439.731,A -85,B 0,C 180,E1 -2105.315,E2 -2105.315} C_VEL
LIN {X 0,Y 573.565,Z 450.498,A -85,B 0,C 180,E1 -2105.81,E2 -2105.81} C_VEL
LIN {X 0,Y 573.49,Z 460.039,A -85,B 0,C 180,E1 -2106.358,E2 -2106.358} C_VEL
LIN {X 0,Y 573.357,Z 469.815,A -85,B 0,C 180,E1 -2107.046,E2 -2107.046} C_VEL
LIN {X 0,Y 573.248,Z 478.74,A -85,B 0,C 180,E1 -2107.807,E2 -2107.807} C_VEL
LIN {X 0,Y 573.195,Z 487.452,A -85,B 0,C 180,E1 -2108.706,E2 -2108.706} C_VEL
LIN {X 0,Y 573.131,Z 494.749,A -85,B 0,C 180,E1 -2109.617,E2 -2109.617} C_VEL
LIN {X 0,Y 573.031,Z 502.269,A -85,B 0,C 180,E1 -2110.775,E2 -2110.775} C_VEL
LIN {X 0,Y 573.035,Z 508.274,A -85,B 0,C 180,E1 -2111.967,E2 -2111.967} C_VEL
LIN {X 0,Y 573.005,Z 512.202,A -85,B 0,C 180,E1 -2112.972,E2 -2112.972} C_VEL
LIN {X 0,Y 572.953,Z 514.27,A -85,B 0,C 180,E1 -2113.638,E2 -2113.638} C_VEL
LIN {X 0,Y 572.966,Z 516.663,A -85,B 0,C 180,E1 -2114.648,E2 -2114.648} C_VEL
LIN {X 0,Y 572.945,Z 518.178,A -85,B 0,C 180,E1 -2115.638,E2 -2115.638} C_VEL
LIN {X 0,Y 572.936,Z 518.88,A -85,B 0,C 180,E1 -2116.612,E2 -2116.612} C_VEL
LIN {X 0,Y 572.99,Z 518.838,A -85,B 0,C 180,E1 -2117.576,E2 -2117.576} C_VEL
LIN {X 0,Y 572.951,Z 518.091,A -85,B 0,C 180,E1 -2118.518,E2 -2118.518} C_VEL
LIN {X 0,Y 572.965,Z 515.576,A -85,B 0,C 180,E1 -2119.942,E2 -2119.942} C_VEL
LIN {X 0,Y 572.965,Z 511.653,A -85,B 0,C 180,E1 -2121.276,E2 -2121.276} C_VEL
LIN {X 0,Y 573.028,Z 506.309,A -85,B 0,C 180,E1 -2122.546,E2 -2122.546} C_VEL
LIN {X 0,Y 573.084,Z 501.158,A -85,B 0,C 180,E1 -2123.503,E2 -2123.503} C_VEL
LIN {X 0,Y 573.095,Z 493.704,A -85,B 0,C 180,E1 -2124.612,E2 -2124.612} C_VEL
LIN {X 0,Y 573.189,Z 486.827,A -85,B 0,C 180,E1 -2125.454,E2 -2125.454} C_VEL
LIN {X 0,Y 573.284,Z 478.47,A -85,B 0,C 180,E1 -2126.308,E2 -2126.308} C_VEL
LIN {X 0,Y 573.373,Z 469.754,A -85,B 0,C 180,E1 -2127.049,E2 -2127.049} C_VEL
LIN {X 0,Y 573.438,Z 459.893,A -85,B 0,C 180,E1 -2127.742,E2 -2127.742} C_VEL
LIN {X 0,Y 573.614,Z 447.931,A -85,B 0,C 180,E1 -2128.413,E2 -2128.413} C_VEL
LIN {X 0,Y 573.707,Z 435.674,A -85,B 0,C 180,E1 -2128.933,E2 -2128.933} C_VEL
LIN {X 0,Y 573.755,Z 423.349,A -85,B 0,C 180,E1 -2129.306,E2 -2129.306} C_VEL
LIN {X 0,Y 573.854,Z 410.704,A -85,B 0,C 180,E1 -2129.554,E2 -2129.554} C_VEL
LIN {X 0,Y 574.051,Z 313.36,A -85,B 0,C 180,E1 -2130.778,E2 -2130.778} C_VEL
LIN {X 0,Y 573.227,Z 308.37,A -85,B 0,C 180,E1 -2130.871,E2 -2130.871} C_VEL
LIN {X 0,Y 573.363,Z 293.801,A -85,B 0,C 180,E1 -2133.483,E2 -2133.483} C_VEL
LIN {X 0,Y 573.405,Z 280.227,A -85,B 0,C 180,E1 -2135.95,E2 -2135.95} C_VEL
LIN {X 0,Y 573.294,Z 279.071,A -85,B 0,C 180,E1 -2136.185,E2 -2136.185} C_VEL
LIN {X 0,Y 573.252,Z 279.082,A -85,B 0,C 180,E1 -2139.173,E2 -2139.173} C_VEL
LIN {X 0,Y 573.223,Z 279.086,A -85,B 0,C 180,E1 -2141.411,E2 -2141.411} C_VEL
LIN {X 0,Y 573.25,Z 279.08,A -85,B 0,C 180,E1 -2143.621,E2 -2143.621} C_VEL
LIN {X 0,Y 573.274,Z 279.075,A -85,B 0,C 180,E1 -2145.807,E2 -2145.807} C_VEL
LIN {X 0,Y 573.265,Z 279.071,A -85,B 0,C 180,E1 -2148.745,E2 -2148.745} C_VEL
LIN {X 0,Y 573.256,Z 279.08,A -85,B 0,C 180,E1 -2151.54,E2 -2151.54} C_VEL
LIN {X 0,Y 573.239,Z 279.084,A -85,B 0,C 180,E1 -2153.665,E2 -2153.665} C_VEL
LIN {X 0,Y 573.224,Z 279.086,A -85,B 0,C 180,E1 -2155.781,E2 -2155.781} C_VEL
LIN {X 0,Y 573.308,Z 279.075,A -85,B 0,C 180,E1 -2157.892,E2 -2157.892} C_VEL
LIN {X 0,Y 573.328,Z 279.062,A -85,B 0,C 180,E1 -2160.702,E2 -2160.702} C_VEL
LIN {X 0,Y 573.301,Z 279.066,A -85,B 0,C 180,E1 -2162.81,E2 -2162.81} C_VEL
LIN {X 0,Y 573.289,Z 279.07,A -85,B 0,C 180,E1 -2165.628,E2 -2165.628} C_VEL
LIN {X 0,Y 573.283,Z 279.074,A -85,B 0,C 180,E1 -2168.459,E2 -2168.459} C_VEL
LIN {X 0,Y 573.273,Z 279.069,A -85,B 0,C 180,E1 -2171.312,E2 -2171.312} C_VEL
LIN {X 0,Y 573.283,Z 279.078,A -85,B 0,C 180,E1 -2174.424,E2 -2174.424} C_VEL
LIN {X 0,Y 573.259,Z 279.071,A -85,B 0,C 180,E1 -2177.112,E2 -2177.112} C_VEL
LIN {X 0,Y 573.243,Z 279.076,A -85,B 0,C 180,E1 -2180.077,E2 -2180.077} C_VEL
LIN {X 0,Y 573.235,Z 279.079,A -85,B 0,C 180,E1 -2182.338,E2 -2182.338} C_VEL
LIN {X 0,Y 573.254,Z 279.073,A -85,B 0,C 180,E1 -2185.41,E2 -2185.41} C_VEL
LIN {X 0,Y 573.248,Z 279.072,A -85,B 0,C 180,E1 -2188.028,E2 -2188.028} C_VEL
LIN {X 0,Y 573.247,Z 279.073,A -85,B 0,C 180,E1 -2190.176,E2 -2190.176} C_VEL
LIN {X 0,Y 573.253,Z 279.076,A -85,B 0,C 180,E1 -2192.645,E2 -2192.645} C_VEL
LIN {X 0,Y 573.207,Z 279.086,A -85,B 0,C 180,E1 -2195.188,E2 -2195.188} C_VEL
LIN {X 0,Y 573.237,Z 279.075,A -85,B 0,C 180,E1 -2197.808,E2 -2197.808} C_VEL
LIN {X 0,Y 573.246,Z 279.073,A -85,B 0,C 180,E1 -2200.525,E2 -2200.525} C_VEL
LIN {X 0,Y 573.239,Z 279.084,A -85,B 0,C 180,E1 -2203.359,E2 -2203.359} C_VEL
LIN {X 0,Y 573.238,Z 279.074,A -85,B 0,C 180,E1 -2206.641,E2 -2206.641} C_VEL
LIN {X 0,Y 573.247,Z 279.083,A -85,B 0,C 180,E1 -2209.475,E2 -2209.475} C_VEL
LIN {X 0,Y 573.236,Z 279.077,A -85,B 0,C 180,E1 -2212.192,E2 -2212.192} C_VEL
LIN {X 0,Y 573.235,Z 279.078,A -85,B 0,C 180,E1 -2215.229,E2 -2215.229} C_VEL
LIN {X 0,Y 573.253,Z 279.083,A -85,B 0,C 180,E1 -2217.772,E2 -2217.772} C_VEL
LIN {X 0,Y 573.265,Z 279.072,A -85,B 0,C 180,E1 -2220.634,E2 -2220.634} C_VEL
LIN {X 0,Y 573.237,Z 279.078,A -85,B 0,C 180,E1 -2223.508,E2 -2223.508} C_VEL
LIN {X 0,Y 573.239,Z 279.085,A -85,B 0,C 180,E1 -2226.135,E2 -2226.135} C_VEL
LIN {X 0,Y 573.269,Z 279.11,A -85,B 0,C 180,E1 -2226.55,E2 -2226.55} C_VEL
LIN {X 0,Y 573.97,Z 284.309,A -85,B 0,C 180,E1 -2227.312,E2 -2227.312} C_VEL
LIN {X 0,Y 573.822,Z 301.466,A -85,B 0,C 180,E1 -2229.757,E2 -2229.757} C_VEL
LIN {X 0,Y 573.605,Z 321.142,A -85,B 0,C 180,E1 -2232.568,E2 -2232.568} C_VEL
LIN {X 0,Y 573.424,Z 343.093,A -85,B 0,C 180,E1 -2235.658,E2 -2235.658} C_VEL
LIN {X 0,Y 573.393,Z 346.611,A -85,B 0,C 180,E1 -2236.149,E2 -2236.149} C_VEL
LIN {X 0,Y 574.07,Z 352.482,A -85,B 0,C 180,E1 -2236.256,E2 -2236.256} C_VEL
LIN {X 0,Y 573.866,Z 454.929,A -85,B 0,C 180,E1 -2237.557,E2 -2237.557} C_VEL
LIN {X 0,Y 573.789,Z 468.207,A -85,B 0,C 180,E1 -2237.869,E2 -2237.869} C_VEL
LIN {X 0,Y 573.675,Z 480.367,A -85,B 0,C 180,E1 -2238.293,E2 -2238.293} C_VEL
LIN {X 0,Y 573.591,Z 492.629,A -85,B 0,C 180,E1 -2238.873,E2 -2238.873} C_VEL
LIN {X 0,Y 573.437,Z 504.195,A -85,B 0,C 180,E1 -2239.585,E2 -2239.585} C_VEL
LIN {X 0,Y 573.329,Z 514.597,A -85,B 0,C 180,E1 -2240.385,E2 -2240.385} C_VEL
LIN {X 0,Y 573.237,Z 523.066,A -85,B 0,C 180,E1 -2241.184,E2 -2241.184} C_VEL
LIN {X 0,Y 573.16,Z 530.958,A -85,B 0,C 180,E1 -2242.071,E2 -2242.071} C_VEL
LIN {X 0,Y 573.075,Z 538.939,A -85,B 0,C 180,E1 -2243.183,E2 -2243.183} C_VEL
LIN {X 0,Y 573.07,Z 545.678,A -85,B 0,C 180,E1 -2244.369,E2 -2244.369} C_VEL
LIN {X 0,Y 573.028,Z 550.371,A -85,B 0,C 180,E1 -2245.427,E2 -2245.427} C_VEL
LIN {X 0,Y 573.022,Z 553.956,A -85,B 0,C 180,E1 -2246.484,E2 -2246.484} C_VEL
LIN {X 0,Y 572.959,Z 555.807,A -85,B 0,C 180,E1 -2247.187,E2 -2247.187} C_VEL
LIN {X 0,Y 572.938,Z 557.197,A -85,B 0,C 180,E1 -2247.891,E2 -2247.891} C_VEL
